S_InterferenceArmElevator2 :=  FaultSim(FaultLow:= VerificationBusyBlockedLow , FaultHigh := VerificationBusyBlockedHigh , Input := VerificationBusy);
S_IsElevatorUp2 :=  FaultSim(FaultLow:=CylinderUpToMeasureLoadBlockedLow  , FaultHigh := CylinderUpToMeasureLoadBlockedHigh , Input := CylinderUpToMeasureLoad);
S_IsElevatorDown2 :=  FaultSim(FaultLow:= CylinderDownToMeasureLoadBlockedLow , FaultHigh := CylinderDownToMeasureLoadBlockedHigh , Input := CylinderDownToMeasureLoad);
S_CylinderRetracted2 :=  FaultSim(FaultLow:= CylinderOfExtractionInRetroactivePositionBlockedLow , FaultHigh := CylinderOfExtractionInRetroactivePositionBlockedHigh , Input := CylinderOfExtractionInRetroactivePosition);
S_CylinderExtended2 :=  FaultSim(FaultLow:= ToExtendCylinderOfExtractionVsGuideBlocked , FaultHigh := ToExtendCylinderOfExtractionVsGuideBlockedHigh , Input := CylinderOfExtractionInExtensivePosition);
S_ElementInElevator2 :=  FaultSim(FaultLow:= ReadyLoadForVerificationBlockedLow , FaultHigh := ReadyLoadForVerificationBlockedHigh , Input := ReadyLoadForVerification);
S_Color2 :=  FaultSim(FaultLow:= ColourMeasurementBlockedLow , FaultHigh := ColourMeasurementBlockedHigh , Input := ColourMeasurement); (* 1 for silver-red element / 0 for black *)
S_IsHigh2 :=  FaultSim(FaultLow:= MeasurementNotOkBlockedLow , FaultHigh := MeasurementNotOkBlockedHigh , Input := MeasurementNotOk);(*1 for high element / 0 for short element*)

(*Sensors of the 3° station*)

S_RotaryAlligned3 :=  FaultSim(FaultLow:= AlignementRotaryTableWithPositioningsBlockedLow , FaultHigh := AlignementRotaryTableWithPositioningsBlockedHigh , Input := AlignementRotaryTableWithPositionings);
S_AvaiableElement3 :=  FaultSim(FaultLow:= AvailableLoadForWorkingStationBlockedLow , FaultHigh := AvailableLoadForWorkingStationBlockedHigh , Input := AvailableLoadForWorkingStation);
S_ControlElement3 :=  FaultSim(FaultLow:= AvailableLoadInControlPositioningBlockedLow , FaultHigh := AvailableLoadInControlPositioningBlockedHigh , Input := AvailableLoadInControlPositioning);
S_DrillElement3 :=  FaultSim(FaultLow:= AvailableLoadInDrillingPositioningBlockedLow , FaultHigh := AvailableLoadInDrillingPositioningBlockedHigh , Input := AvailableLoadInDrillingPositioning);
S_IsOnTheRightSide3 :=  FaultSim(FaultLow:= InControlLoadInWrongPositionToBeDrilledBlockedLow , FaultHigh := InControlLoadInWrongPositionToBeDrilledBlockedHigh , Input := InControlLoadInWrongPositionToBeDrilled);
S_DrillUp3 :=  FaultSim(FaultLow:= DrillingUnitUpBlockedLow , FaultHigh := DrillingUnitUpBlockedHigh , Input := DrillingUnitUp);
S_DrillDown3 :=  FaultSim(FaultLow:= DrillingUnitDownBlockedLow , FaultHigh := DrillingUnitDownBlockedHigh , Input := DrillingUnitDown);

(*Sensors of the 4° station*)

S_SpringCylinderExtended4 :=  FaultSim(FaultLow:= ToExtractSpringInAssemblyStationInExtensivePositionBlockedLow , FaultHigh := ToExtractSpringInAssemblyStationInExtensivePositionBlockedHigh , Input := ToExtractSpringInAssemblyStationInExtensivePosition);
S_SpringCylinderRetracted4 :=  FaultSim(FaultLow:= ToExtractSpringInAssemblyStationInRetroactivePositionBlockedLow , FaultHigh := ToExtractSpringInAssemblyStationInRetroactivePositionBlockedHigh , Input := ToExtractSpringInAssemblyStationInRetroactivePosition);
S_BlackPistonGiven4 :=  FaultSim(FaultLow:= PistonSelectorIsOnTheRightBlockedLow , FaultHigh := PistonSelectorIsOnTheRightBlockedHigh , Input := PistonSelectorIsOnTheRight);
S_SilverPistonGiven4 :=  FaultSim(FaultLow:= PistonSelectorIsOnTheLeftBlockedLow , FaultHigh := PistonSelectorIsOnTheLeftBlockedHigh , Input := PistonSelectorIsOnTheLeft);
S_NoCover4 :=  FaultSim(FaultLow:= EmptyCoverHouseInAssemblyStationBlockedLow , FaultHigh := EmptyCoverHouseInAssemblyStationBlockedHigh , Input := EmptyCoverHouseInAssemblyStation);
S_CoverCylinderRetracted4 :=  FaultSim(FaultLow:= ToExtractCoverInAssemblyStationInRetroactivePositionBlockedLow , FaultHigh := ToExtractCoverInAssemblyStationInRetroactivePositionBlockedHigh , Input := ToExtractCoverInAssemblyStationInRetroactivePosition);
S_CoverCylinderExtracted4 :=  FaultSim(FaultLow:= ToExtractCoverInAssemblyStationInExtensivePositionBlockedLow , FaultHigh := ToExtractCoverInAssemblyStationInExtensivePositionBlockedHigh , Input := ToExtractCoverInAssemblyStationInExtensivePosition);
S_ElementAvailable4 :=  FaultSim(FaultLow:= AvailableLoadForRobotBlockedLow , FaultHigh := AvailableLoadForRobotBlockedHigh , Input := AvailableLoadForRobot);

(*Robot sensors simulation*)

RobotInInitialPosition := Bit0Input AND Bit1Input;
RobotInAssemblyUnit := Bit3Input;
RobotInPistonWarehouse := Bit0Input AND NOT Bit1Input;
RobotInSpringWarehouse := NOT Bit0Input AND Bit1Input;
RobotInCoverWarehouse := Bit2Input;

S_RobotInInitial4 :=  FaultSim(FaultLow:= RobotInInitialPositionBlockedLow , FaultHigh := RobotInInitialPositionBlockedHigh , Input := RobotInInitialPosition);
S_RobotAssembly4 :=  FaultSim(FaultLow:= RobotInAssemblyUnitBlockedLow , FaultHigh := RobotInAssemblyUnitBlockedHigh , Input := RobotInAssemblyUnit);
S_RobotPiston4 :=  FaultSim(FaultLow:= RobotInPistonWarehouseBlockedLow , FaultHigh := RobotInPistonWarehouseBlockedHigh , Input := RobotInPistonWarehouse);
S_RobotSpring4 :=  FaultSim(FaultLow:= RobotInSpringWarehouseBlockedLow , FaultHigh := RobotInSpringWarehouseBlockedHigh , Input := RobotInSpringWarehouse);
S_RobotCover4 :=  FaultSim(FaultLow:= RobotInCoverWarehouseBlockedLow , FaultHigh := RobotInCoverWarehouseBlockedHigh , Input := RobotInCoverWarehouse);


(*Buttons*)

B_Start := Start;
B_Reset := Reset;
B_Freeze := NOT FreezeStopPuls;
B_Stop := NOT Stop;
B_Emergency := NOT EmergencyStop;
B_FullWarehouse := FullWarehouse;
B_OnlyBlackElement := ToWorkBlackLoad; (*1 to work only on black elements / 0 to work only on red/silver elements*)
B_AllColors := ToWorkBlackOrRedLoad; (*1 all colors / 0 only one color check B_OnlyBlackElement*)
B_FaultyElementRemoved := UpsideDownLoadRemovedInExpelling;
B_FillAll := FillAllWarehouses;
END_PROGRAM

(* POU Bridge/FaultSim, ST *)
FUNCTION FaultSim : BOOL

VAR_INPUT

	FaultLow: BOOL;
	FaultHigh: BOOL;
	Input: BOOL;

END_VAR

VAR
END_VAR
IF FaultLow THEN
	FaultSim := FALSE;
ELSIF FaultHigh THEN
	FaultSim := TRUE;
ELSE
	FaultSim := Input;
END_IF
END_FUNCTION

(* POU Main, ST *)
PROGRAM Main

VAR

	Stazione1: S1;
	Stazione2: S2;
	Stazione3: S3;
	Stazione4: S4;
	Lights: Lights;
	InitializationDone: BOOL := FALSE;
	ElementS2: CharacterisazionElement;
	ElementS3: CharacterisazionElement;
	ElementS4: CharacterisazionElement;
	OperationType: INT := INIT;
	Station1OperationType: INT := INIT;
	Station2OperationType: INT := INIT;
	Station3OperationType: INT := INIT;
	Station4OperationType: INT := INIT;
	NotSafeToRestart: BOOL;
	OnPhaseStopDone: BOOL;
	StopDone: BOOL;
	FirstPowerOn : BOOL := TRUE;
	RunCycles: INT := 0; (* Debug Variable used to take time-measurements *)

END_VAR
IF (OperationType = INIT) THEN
	SignHandlerOperationType := INIT;
ELSE
	SignHandlerOperationType := RUN;
END_IF

SignalHandler();

IF EmergencyInStop THEN

	OperationType := EMERGENCYSTOPMACHINE;
	Station1OperationType := IMMEDIATESTOPMACHINE; (*In emergency operation type Stations act as in the immediate stop case*)
	Station2OperationType := IMMEDIATESTOPMACHINE;
	Station3OperationType := IMMEDIATESTOPMACHINE;
	Station4OperationType := IMMEDIATESTOPMACHINE;
	Stazione1.StartButton := FALSE;

END_IF

CASE OperationType OF

	INIT:

		BridgeInitOperation := TRUE; (* Used only for Real Plant *)
		IF NOT MachineNOTOkForReset THEN		(* After a Reset it is FALSE, but not for first POWER-ON *)

			FirstPowerOn := FALSE;
			LightMachineToBeEmpty := FALSE;
			ButtonMachineToBeEmptyInvisible := TRUE;
			Station1OperationType := INIT;
			Station2OperationType := INIT;
			Station3OperationType := INIT;
			Station4OperationType := INIT;

		END_IF

		IF  Stazione1.InitializationDone1 AND  Stazione2.InitializationDone2 AND Stazione3.InitializationDone3  AND Stazione4.InitializationDone4  THEN (*Wait all station initialized*)
			InitializationDone:=TRUE;
			OperationType := READYTORUN;
		END_IF

	READYTORUN: (* Idle State*)

		BridgeInitOperation := FALSE; (* Used only for Real Plant *)
		Station1OperationType := READYTORUN;
		Station2OperationType := READYTORUN;
		Station3OperationType := READYTORUN;
		Station4OperationType := READYTORUN;

		IF B_Start THEN

			MachineNOTOkForReset := TRUE;
			LightMachineToBeEmpty := TRUE;
			OperationType:= RUN;
			Stazione1.StartButton := TRUE;

		END_IF

	RUN:

		RunCycles := RunCycles +1; (* For Diagnostic *)

		Station1OperationType := RUN;
		Station2OperationType := RUN;
		Station3OperationType := RUN;
		Station4OperationType := RUN;

		Stazione1.Go:= Stazione2.GoS1; (*To NOT have interference between stations *) (* Station(i+1) communicate when Station(i) can go i= 1,2,3 *)
		Stazione2.Go:= Stazione3.GoS2;
		Stazione3.Go:= Stazione4.GoS3;

		ElementS2.Color:=Stazione2.ActualColor;
		ElementS3.Over:=Stazione3.PieceOverturned;
		Stazione4.ElementColor:= ElementS4.Color;
		Stazione4.ElementOver:= ElementS4.Over;

		IF Stazione2.PassElementDefinition THEN (*Station(i) communicate the characterization of the piece done to Station(i+1) i= 2,3*)
			ElementS3.Color := ElementS2.Color;
		END_IF

		IF Stazione3.PassElementDefinition THEN
			ElementS4.Color := ElementS3.Color;
			ElementS4.Over := ElementS3.Over;
		END_IF

		IF ImmediateInStop THEN

			OperationType := IMMEDIATESTOPMACHINE;
			Station1OperationType := IMMEDIATESTOPMACHINE;
			Station2OperationType := IMMEDIATESTOPMACHINE;
			Station3OperationType := IMMEDIATESTOPMACHINE;
			Station4OperationType := IMMEDIATESTOPMACHINE;
			Stazione1.StartButton := FALSE;

		END_IF

		IF OnPhaseInStop THEN

			OperationType := ONPHASESTOPMACHINE;
			Station1OperationType := ONPHASESTOPMACHINE;
			Station2OperationType := ONPHASESTOPMACHINE;
			Station3OperationType := ONPHASESTOPMACHINE;
			Station4OperationType := ONPHASESTOPMACHINE;
			Stazione1.StartButton := FALSE;

		END_IF

	IMMEDIATESTOPMACHINE:

		IF NOT ImmediateInStop AND StopDone THEN  (* Wait until all the stations stop*)
			IF NotSafeToRestart  THEN
				OperationType := READYTORESET;
			ELSE
				OperationType := READYTORUN;
			END_IF
		END_IF


	ONPHASESTOPMACHINE:

		IF OnPhaseStopDone THEN (* Wait until all the stations stop*)
			OperationType := READYTORUN;
		END_IF

	EMERGENCYSTOPMACHINE:

		IF StopDone THEN (* Wait until all the stations stop*)
			OperationType := READYTORESET;
		END_IF

	READYTORESET:

		ButtonMachineToBeEmptyInvisible := FALSE;
		LightMachineToBeEmpty := TRUE;
		Station1OperationType := READYTORESET;
		Station2OperationType := READYTORESET;
		Station3OperationType := READYTORESET;
		Station4OperationType := READYTORESET;

		IF B_Reset AND NOT(ImmediateInStop OR EmergencyInStop OR NOT NoSignalsToReset OR MachineNOTOkForReset)  THEN
			InitializationDone := FALSE;
			OperationType := INIT;
		END_IF

END_CASE

AllStationsIdle := (	Stazione1.Idle AND Stazione2.Idle AND Stazione3.Idle AND Stazione4.Idle AND  (OperationType=RUN));	(* Signal Used to Stop Machine for inactivity*)
NotSafeToRestart := Stazione1.NotSafeToRestart OR Stazione2.NotSafeToRestart OR Stazione3.NotSafeToRestart OR Stazione4.NotSafeToRestart;
OnPhaseStopDone := Stazione1.OnPhaseStopDone1 AND Stazione2.OnPhaseStopDone2 AND Stazione3.OnPhaseStopDone3 AND Stazione4.OnPhaseStopDone4;
StopDone := Stazione1.StopDone1 AND Stazione2.StopDone2 AND Stazione3.StopDone3 AND Stazione4.StopDone4;

(*Update calls*)

ClocksGeneration.OperationType:= OperationType;
ClocksGeneration();

Lights.OperationType:= OperationType;
Lights.Element2.Color := ElementS2.Color;
Lights.Element3.Color := ElementS3.Color;
Lights.Element3.Over := Stazione3.PieceOverturned;
Lights.WriteLight2 := NOT Stazione2.GoS1;
Lights.WriteLight3 := Stazione3.WriteLight;
Lights.WriteLight4 := NOT Stazione4.Idle;
Lights.Element4 := Stazione4.Element;
Lights.InitializationDone:=InitializationDone;
Lights.RobotMoving := Stazione4.RobotIsMoving;
Lights.RobotOn := Stazione4.RobotIsOn;
Lights.PieceToDiscard2 := Stazione2.PieceToDiscard2;
Lights.Rejected:=Stazione4.Rejected;
Lights.Completed:=Stazione4.Completed;

 IF ClocksGeneration.Clock2ms AND NOT FirstPowerOn THEN
Lights();
Stazione1(OperationType := Station1OperationType);
Stazione2(OperationType := Station2OperationType);
Stazione3(OperationType := Station3OperationType);
Stazione4(OperationType := Station4OperationType);
 END_IF
END_PROGRAM

(* POU Work_Station/S1, ST *)
(* @OBJECTFLAGS := '0, 8' *)

FUNCTION_BLOCK S1

VAR_INPUT

	StartButton : BOOL;
	Go : BOOL;

END_VAR

VAR_OUTPUT

	InitializationDone1: BOOL;
	OnPhaseStopDone1: BOOL := FALSE;
	StopDone1: BOOL := FALSE;
	NotSafeToRestart: BOOL;
	Idle: BOOL;

END_VAR

VAR

	Cylinder: GenericDevice;
	Rotary : GenericDevice;
	Vacuum :GenericDevice;
	Expulsion :GenericDevice;
	EnableRotary: BOOL := FALSE;
	DisableRotary: BOOL:= FALSE;
	StateMachine: INT;
	EnableCylinder: BOOL := FALSE;
	DisableCylinder: BOOL := FALSE;
	EnableVacuum: BOOL := FALSE;
	DisableVacuum: BOOL := FALSE;
	EnableExpulsion: BOOL := FALSE;
	DisableExpulsion: BOOL := FALSE;
	NextElementReady: BOOL;
	CylinderInitialized: BOOL := FALSE;
	RotaryInitialized: BOOL := FALSE;
	VacuumInitialized: BOOL := FALSE;
	ExpulsionInitialized: BOOL := FALSE;
	ActivateVacuum: BOOL := FALSE;
	ActivateExpulsion: BOOL := FALSE;

END_VAR

VAR_IN_OUT

	OperationType: INT;

END_VAR
CASE OperationType OF

	INIT:

		IF CylinderInitialized AND RotaryInitialized AND VacuumInitialized AND ExpulsionInitialized THEN (* Wait until all devices are initialized*)
			InitializationDone1 := TRUE;
		END_IF

	READYTORUN:

		NotSafeToRestart := FALSE;
		OnPhaseStopDone1 := FALSE;
		StopDone1 := FALSE;

	RUN:

		IF ActivateVacuum THEN (*To safely restart after an immediate stop*)
			EnableVacuum := TRUE;
			ActivateVacuum := FALSE;
		END_IF

		IF ActivateExpulsion THEN (*To safely restart after an immediate stop*)
			EnableExpulsion := TRUE;
			ActivateExpulsion := FALSE;
		END_IF

		CASE StateMachine OF

			0: (*Wait Start button*)
				IF StartButton THEN
					StateMachine := 1;
				END_IF

			1:
				DisableCylinder := TRUE;
				StateMachine := 5;

			5: (*With no interference with the elevator the rotary can turn*)

				Idle:=TRUE;

				IF NOT DisableCylinder AND  NOT S_EmptyWarehouse1 AND Go THEN
					Idle:=FALSE;
					DisableRotary:=TRUE;
					StateMachine :=10;
				END_IF

			10: (*Moving the element with the cylinder*)

				IF NOT DisableRotary THEN
					EnableCylinder := TRUE;
					StateMachine := 15;
				END_IF

			15: (*Turn rotary*)

				IF NOT EnableCylinder  THEN
					EnableRotary := TRUE;
					StateMachine := 20;
				END_IF

			20: (*Activation vacuum*)

				IF NOT EnableRotary THEN
					EnableVacuum := TRUE;
					StateMachine := 25;
				END_IF

			25: (*Move Rotary to station 2 and cylinder retracts*)

				IF NOT EnableVacuum AND Go THEN
					DisableRotary := TRUE;
					DisableCylinder := TRUE;
					StateMachine := 30;
				END_IF

			30: (*Disable vacuum *)

				IF NOT DisableRotary AND  NOT DisableCylinder AND NOT ActivateVacuum THEN
					DisableVacuum := TRUE;
					IF NOT S_EmptyWarehouse1 THEN (*If there is a piece available the cylinder ejects it before enabling the rotary*)
						EnableCylinder:=TRUE;
						NextElementReady := TRUE;
					ELSE
						NextElementReady := FALSE;
					END_IF

					StateMachine := 35;
				END_IF

			35: (*Expell the element from the suction cup *)

				IF (NOT DisableVacuum AND NOT NextElementReady) OR (NOT DisableVacuum AND NOT EnableCylinder AND NextElementReady) THEN
					EnableExpulsion := TRUE;
					StateMachine := 40;
				END_IF

			40: (*Move  the rotary to warehouse*)

				IF NOT EnableExpulsion THEN
					DisableExpulsion:=TRUE;
					EnableRotary := TRUE;
					StateMachine := 50;
				END_IF

			50: (*Go back to the initial state*)

				IF NOT EnableRotary AND NOT DisableExpulsion THEN
					IF NextElementReady THEN
						StateMachine:=20;
					ELSE
						StateMachine := 5;
					END_IF
				END_IF

	END_CASE

	IMMEDIATESTOPMACHINE:

		CASE StateMachine OF
			0:
				StopDone1 := TRUE;

			1:
				StopDone1 := TRUE;

			5:
				IF NOT DisableCylinder THEN
					StopDone1 := TRUE;
				END_IF

			10:
				IF NOT DisableRotary THEN
					StopDone1 := TRUE;
				END_IF

			15:
				IF NOT EnableCylinder  THEN
					StopDone1 := TRUE;
				END_IF

			20:
				IF NOT EnableRotary THEN
					StopDone1 := TRUE;
				END_IF

			25:
				DisableVacuum := TRUE;
				ActivateVacuum := TRUE;
				StopDone1 := TRUE;

			30:
				IF NOT DisableRotary AND  NOT DisableCylinder THEN
					DisableVacuum := TRUE;
					StopDone1 := TRUE;
				END_IF

			35:
				IF (NOT DisableVacuum AND NOT NextElementReady) OR (NOT DisableVacuum AND NOT EnableCylinder AND NextElementReady) THEN
					StopDone1 := TRUE;
				END_IF

			40:
				DisableExpulsion := TRUE;
				ActivateExpulsion := TRUE;
				StopDone1 := TRUE;

			50:
				IF NOT EnableRotary AND NOT DisableExpulsion THEN
					StopDone1 := TRUE;
				END_IF

	END_CASE

	ONPHASESTOPMACHINE:

		CASE StateMachine OF

			0:
				OnPhaseStopDone1 := TRUE;

			1:
				OnPhaseStopDone1 := TRUE;

			5:
				IF NOT DisableCylinder THEN
					OnPhaseStopDone1 := TRUE;
				END_IF

			10:
				IF NOT DisableRotary THEN
					OnPhaseStopDone1 := TRUE;
				END_IF

			15:
				IF NOT EnableCylinder  THEN
					OnPhaseStopDone1 := TRUE;
				END_IF

			20:
				IF NOT EnableRotary THEN
					OnPhaseStopDone1 := TRUE;
				END_IF

			25:
				IF NOT EnableVacuum THEN
					OnPhaseStopDone1 := TRUE;
				END_IF

			30:
				IF NOT DisableRotary AND  NOT DisableCylinder THEN
					DisableVacuum := TRUE;
					OnPhaseStopDone1 := TRUE;
				END_IF

			35:
				IF (NOT DisableVacuum AND NOT NextElementReady) OR (NOT DisableVacuum AND NOT EnableCylinder AND NextElementReady) THEN
					OnPhaseStopDone1 := TRUE;
				END_IF

			40:
				IF NOT EnableExpulsion THEN
					OnPhaseStopDone1 := TRUE;
				END_IF

			50:
				IF NOT EnableRotary AND NOT DisableExpulsion THEN
					OnPhaseStopDone1 := TRUE;
				END_IF
	END_CASE


	READYTORESET:

		InitializationDone1 := FALSE;
		StateMachine := 0;
		ActivateVacuum := FALSE;
		ActivateExpulsion := FALSE;

END_CASE

(*Cylinder Generic Device*)

Cylinder(DeviceEnableRequest:=EnableCylinder ,DeviceDisableRequest := DisableCylinder);
A_Cylinder1 := Cylinder.EnableDevice;
Cylinder.DeviceEnabled  := S_CylinderExtended1;
Cylinder.DeviceDisabled := S_CylinderRetracted1;
Cylinder.DeviceType := DEVICE_WITH_SINGLE_ACTUATION OR DEVICE_WITH_DOUBLE_FEEDBACK;
Cylinder.DeviceClock := ClocksGeneration.Clock2ms;
Cylinder.DeviceDiagnosticsEnabled := TRUE;
Cylinder.DeviceDisableTime := 20;
Cylinder.DeviceEnablePreset := TRUE;
Cylinder.DeviceEnableTime := 20;
Cylinder.DeviceOperation := OperationType;
CylinderInitialized := NOT Cylinder.DeviceNotInitialized;
F_Cylinder1 := Cylinder.DeviceFault;
F_S_Cylinder1 := Cylinder.DeviceSensorFault;
F_A_Cylinder1 := Cylinder.DeviceActuatorFault;
FH_A_Cylinder1 := Cylinder.DeviceActuatorFaultHigh;
FL_A_Cylinder1 := Cylinder.DeviceActuatorFaultLow;
FH_DS_Cylinder1 := Cylinder.DeviceDisabledSensorFaultHigh;
FL_DS_Cylinder1 := Cylinder.DeviceDisabledSensorFaultLow;
FH_ES_Cylinder1 := Cylinder.DeviceEnabledSensorFaultHigh;
FL_ES_Cylinder1 := Cylinder.DeviceEnabledSensorFaultLow;

(*Rotary Generic Device*)

Rotary(DeviceEnableRequest:=EnableRotary ,DeviceDisableRequest := DisableRotary);
A_ArmToElevator1 := Rotary.DisableDevice;
A_ArmToWarehouse1 := Rotary.EnableDevice;
Rotary.DeviceEnabled := S_ArmInWarehouse1;
Rotary.DeviceDisabled := S_ArmInElevator1;
Rotary.DeviceType := DEVICE_WITH_DOUBLE_FEEDBACK  OR DEVICE_WITH_DOUBLE_ACTUATION;
Rotary.DeviceClock := ClocksGeneration.Clock2ms;
Rotary.DeviceDiagnosticsEnabled := TRUE;
Rotary.DeviceDisableTime := 20;
Rotary.DeviceEnablePreset := TRUE;
Rotary.DeviceEnableTime := 20;
Rotary.DeviceOperation := OperationType;
RotaryInitialized := NOT Rotary.DeviceNotInitialized;
F_Rotary1 := Rotary.DeviceFault;
F_S_Rotary1 := Rotary.DeviceSensorFault;
F_A_Rotary1 := Rotary.DeviceActuatorFault;
FL_EA_Rotary1 := Rotary.DeviceEnableActuatorFaultLow;
FH_EA_Rotary1 := Rotary.DeviceEnableActuatorFaultHigh;
FL_DA_Rotary1 := Rotary.DeviceDisableActuatorFaultLow;
FH_DA_Rotary1 := Rotary.DeviceDisableActuatorFaultHigh;
FH_ES_Rotary1 := Rotary.DeviceEnabledSensorFaultHigh;
FL_ES_Rotary1 := Rotary.DeviceEnabledSensorFaultLow;
FH_DS_Rotary1 := Rotary.DeviceDisabledSensorFaultHigh;
FL_DS_Rotary1 := Rotary.DeviceDisabledSensorFaultLow;

(*Vacuum Generic Device*)

Vacuum(DeviceEnableRequest:=EnableVacuum ,DeviceDisableRequest := DisableVacuum);
Vacuum.DeviceEnabled:= S_VacuumOk1;
A_Vacuum1 := Vacuum.EnableDevice;
Vacuum.DeviceType := DEVICE_WITH_SINGLE_ACTUATION OR DEVICE_WITH_ENABLE_FEEDBACK;
Vacuum.DeviceClock := ClocksGeneration.Clock2ms;
Vacuum.DeviceDiagnosticsEnabled := TRUE;
Vacuum.DeviceDisableTime := 10;
Vacuum.DeviceEnablePreset := FALSE;
Vacuum.DeviceEnableTime := 10;
Vacuum.DeviceOperation := OperationType;
VacuumInitialized := NOT Vacuum.DeviceNotInitialized;
F_Vacuum1 := Vacuum.DeviceFault;
F_S_Vacuum1 := Vacuum.DeviceSensorFault;
F_A_Vacuum1 := Vacuum.DeviceActuatorFault OR Vacuum.DeviceEnabledSensorFault	(* CHECK *);
FH_A_Vacuum1 := Vacuum.DeviceActuatorFaultHigh;
FL_A_Vacuum1 := Vacuum.DeviceEnabledSensorFault;
FH_S_Vacuum1 := Vacuum.DeviceSensorFaultHigh;
FL_S_Vacuum1 := Vacuum.DeviceSensorFaultLow;

(*Expulsion Generic Device*)

Expulsion(DeviceEnableRequest:=EnableExpulsion ,DeviceDisableRequest := DisableExpulsion);
A_AirVacuum1 := Expulsion.EnableDevice;
Expulsion.DeviceType := DEVICE_WITH_SINGLE_ACTUATION OR DEVICE_WITHOUT_FEEDBACK;
Expulsion.DeviceClock := ClocksGeneration.Clock2ms;
Expulsion.DeviceDiagnosticsEnabled := TRUE;
Expulsion.DeviceDisableTime := 10;
Expulsion.DeviceEnablePreset := FALSE;
Expulsion.DeviceEnableTime := 10;
Expulsion.DeviceOperation := OperationType;
ExpulsionInitialized := NOT Expulsion.DeviceNotInitialized;
F_Expulsion1 := Expulsion.DeviceFault;

(* THINK DIAGNOSIS *)

FH_A_Expulsion1 := Expulsion.DeviceActuatorFaultHigh;
FL_A_Expulsion1 := Expulsion.DeviceActuatorFaultLow;
END_FUNCTION_BLOCK

(* POU MyLibraries/GenericDevice, ST *)
FUNCTION_BLOCK GenericDevice

	VAR_INPUT

		DeviceEnableTime : UINT;
		DeviceDisableTime : UINT;
		DeviceEnabled : BOOL;
		DeviceDisabled : BOOL;
		DeviceClock : BOOL;
		DeviceType : BYTE;
		DeviceEnablePreset : BOOL;
		DeviceOperation : INT;
		DeviceDiagnosticsEnabled: BOOL;

END_VAR

	VAR_OUTPUT

		EnableDevice : BOOL;
		DisableDevice : BOOL;

		DeviceDisabledSensorFaultLow : BOOL;
		DeviceDisabledSensorFaultHigh : BOOL;
		DeviceEnabledSensorFaultLow: BOOL;
		DeviceEnabledSensorFaultHigh : BOOL;
		DeviceEnableActuatorFaultLow: BOOL;
		DeviceEnableActuatorFaultHigh : BOOL;
		DeviceDisableActuatorFaultLow : BOOL;
		DeviceDisableActuatorFaultHigh : BOOL;

		DeviceActuatorFaultHigh : BOOL;
		DeviceActuatorFaultLow : BOOL;
		DeviceSensorFaultHigh : BOOL;
		DeviceSensorFaultLow : BOOL;

		DeviceSensorFault : BOOL;
		DeviceActuatorFault : BOOL;
		DeviceFault : BOOL;
		DeviceDisabledSensorFault : BOOL;
		DeviceEnabledSensorFault : BOOL;
		(* End of Diagnostic Internal Variables *)

		DeviceNotInitialized : BOOL;

	END_VAR

	VAR_IN_OUT

		DeviceEnableRequest : BOOL;
		DeviceDisableRequest : BOOL;

	END_VAR

	VAR

		DeviceState : DeviceStateType := 0;
		DeviceTimer : UINT := 0;
		Timeout : BOOL;

	END_VAR

	VAR_EXTERNAL

	(*Feedback*)

	DEVICE_WITHOUT_FEEDBACK : BYTE := 2#01000000;
	DEVICE_WITH_ENABLE_FEEDBACK : BYTE := 2#00010000;
	DEVICE_WITH_DISABLE_FEEDBACK : BYTE := 2#00100000;
	DEVICE_WITH_DOUBLE_FEEDBACK : BYTE := 2#00110000;
	DEVICE_FEEDBACK_MASK : BYTE := 2#11110000;

	(*Actuation*)

	DEVICE_WITH_SINGLE_ACTUATION : BYTE := 2#00000001;
	DEVICE_WITH_DOUBLE_ACTUATION : BYTE := 2#00000011;
	DEVICE_WITH_DA_NO_RETAIN : BYTE := 2#00000010;
	DEVICE_ACTUATION_MASK : BYTE := 2#00001111;

	END_VAR
(*** DEVICE CLOCK HANDLER ***)

IF DeviceClock AND (DeviceTimer > 0) THEN

	DeviceTimer := DeviceTimer - 1;

END_IF;

Timeout := (DeviceTimer = 0);


(*** DEVICE INITIALIZATION HANDLER ***)

IF (DeviceOperation = INIT) THEN

	DeviceEnableRequest := FALSE;
	DeviceDisableRequest := FALSE;

	IF DeviceEnablePreset THEN
		EnableDevice := TRUE;
		DeviceTimer := DeviceEnableTime;

		IF (NOT (DeviceDisabled AND DeviceEnabled)) THEN
			DeviceState := DeviceEnablePhaseState;
		ELSE
			DeviceState := DeviceEnabledState;
		END_IF;
		DeviceNotInitialized := NOT DeviceEnabled OR DeviceDisabled;
	ELSE
		EnableDevice := FALSE;
		DeviceTimer := DeviceDisableTime;
		IF (NOT (DeviceDisabled AND DeviceEnabled)) THEN
			DeviceState := DeviceDisablePhaseState;
		ELSE
			DeviceState := DeviceDisabledState;
		END_IF;
		DeviceNotInitialized := DeviceEnabled OR NOT DeviceDisabled;
	END_IF;

	CASE (DeviceType AND DEVICE_FEEDBACK_MASK) OF

		DEVICE_WITH_ENABLE_FEEDBACK:
			DeviceDisabled := NOT DeviceEnabled;

		DEVICE_WITH_DISABLE_FEEDBACK :
			DeviceEnabled := NOT DeviceDisabled;

		DEVICE_WITHOUT_FEEDBACK:
			DeviceEnabled := DeviceEnablePreset;
			DeviceDisabled := NOT DeviceEnabled;

	END_CASE;

	CASE (DeviceType AND DEVICE_ACTUATION_MASK) OF

		DEVICE_WITH_DOUBLE_ACTUATION:
			DisableDevice := NOT EnableDevice;

		DEVICE_WITH_DA_NO_RETAIN: (* Not sure *)
			EnableDevice := EnableDevice AND (DeviceState = DeviceEnablePhaseState);
			DisableDevice := NOT EnableDevice AND (DeviceState = DeviceDisablePhaseState);

	END_CASE;
ELSE

	(*** DEVICE SENSORS HANDLER ***)

	(*Device with single actuation and single disable feedback*)

	IF (DeviceType AND DEVICE_FEEDBACK_MASK) = DEVICE_WITH_DISABLE_FEEDBACK THEN
		DeviceEnabled := NOT DeviceDisabled AND ((DeviceState = DeviceEnabledState) OR (DeviceState = DeviceEnablePhaseState) AND Timeout);
	END_IF;

	(*Device with single actuation and single enable feedback*)

	IF (DeviceType AND DEVICE_FEEDBACK_MASK) = DEVICE_WITH_ENABLE_FEEDBACK THEN
		DeviceDisabled := NOT DeviceEnabled AND ((DeviceState = DeviceDisabledState) OR (DeviceState = DeviceDisablePhaseState) AND Timeout);
	END_IF;

	(*Device with single actuation and NO feedback*)

	IF (DeviceType AND DEVICE_FEEDBACK_MASK) = DEVICE_WITHOUT_FEEDBACK THEN

		DeviceEnabled :=( (DeviceState = DeviceEnabledState) OR (DeviceState = DeviceEnablePhaseState)) AND Timeout;

		DeviceDisabled := (DeviceState = DeviceDisabledState) OR (DeviceState = DeviceDisablePhaseState) AND Timeout;

	END_IF;


	(*** DEVICE ACTUATORS HANDLER ***)

	(* Device with double actuation*)

	IF (DeviceType AND DEVICE_ACTUATION_MASK) = DEVICE_WITH_DOUBLE_ACTUATION THEN

		DisableDevice := NOT EnableDevice;

	END_IF;

	(* Device with double actuation and NO retain *)

	IF (DeviceType AND DEVICE_ACTUATION_MASK) = DEVICE_WITH_DA_NO_RETAIN THEN

		EnableDevice := EnableDevice AND (DeviceState = DeviceEnablePhaseState);

		DisableDevice := NOT EnableDevice AND (DeviceState = DeviceDisablePhaseState);

	END_IF;

END_IF;


(*** DEVICE CONTROL HANDLER ***)

CASE DeviceState OF

	DeviceDisabledState:

		DeviceDisableRequest := FALSE;

		IF DeviceEnableRequest THEN

			EnableDevice := TRUE;
			DeviceTimer := DeviceEnableTime;
			DeviceState := DeviceEnablePhaseState;

		END_IF;

	DeviceEnablePhaseState:

		IF DeviceDisableRequest THEN

			DeviceEnableRequest := FALSE;
			EnableDevice := FALSE;
			DeviceTimer := DeviceDisableTime;
			DeviceState := DeviceDisablePhaseState;

		END_IF;

		IF DeviceEnabled THEN

			DeviceEnableRequest := FALSE;
			DeviceTimer := 0;
			DeviceState := DeviceEnabledState;

		END_IF;

	DeviceEnabledState:

		DeviceEnableRequest := FALSE;

		IF DeviceDisableRequest THEN

			EnableDevice := FALSE;
			DeviceTimer := DeviceDisableTime;
			DeviceState := DeviceDisablePhaseState;

		END_IF;

	DeviceDisablePhaseState:

		IF DeviceEnableRequest THEN

			DeviceDisableRequest := FALSE;
			EnableDevice := TRUE;
			DeviceTimer := DeviceEnableTime;
			DeviceState := DeviceEnablePhaseState;

		END_IF;

		IF DeviceDisabled THEN

			DeviceDisableRequest := FALSE;
			DeviceTimer := 0;
			DeviceState := DeviceDisabledState;

		END_IF;

END_CASE;

(*** DEVICE DIAGNOSTICS HANDLER ***)

IF DeviceDiagnosticsEnabled THEN

	(* CHECKS HIGH/LOW FAULTS FOR DOUBLE FEEDBACK/ACTUATION TYPES **)

	DeviceDisabledSensorFaultLow := (NOT EnableDevice AND NOT DeviceDisabled AND NOT DeviceEnabled AND ((DeviceState=DeviceDisabledState) OR (DeviceState=DeviceDisablePhaseState))) AND Timeout;	(* FOR DOUBLE FEEDBACK TYPE *)
	DeviceDisabledSensorFaultHigh := (EnableDevice AND DeviceDisabled AND DeviceEnabled AND (DeviceState=DeviceEnabledState)) AND Timeout;					(* FOR DOUBLE FEEDBACK TYPE *)
	DeviceEnabledSensorFaultHigh := (NOT EnableDevice AND DeviceDisabled AND DeviceEnabled AND (DeviceState=DeviceDisabledState)) AND Timeout;				(* FOR DOUBLE FEEDBACK TYPE *)
	DeviceEnabledSensorFaultLow := (EnableDevice AND NOT DeviceDisabled AND NOT DeviceEnabled AND ((DeviceState=DeviceEnablePhaseState) OR (DeviceState=DeviceEnabledState)) ) AND Timeout;			(* FOR DOUBLE FEEDBACK TYPE *)

	DeviceEnableActuatorFaultLow := (EnableDevice AND DeviceDisabled AND NOT DeviceEnabled  AND (DeviceState = DeviceEnablePhaseState)) AND Timeout;		(* FOR DOUBLE ACTUATION TYPE *)
	DeviceEnableActuatorFaultHigh := (NOT EnableDevice AND NOT DeviceDisabled AND DeviceEnabled AND DeviceState = (DeviceDisabledState)) AND Timeout;		(* FOR DOUBLE ACTUATION TYPE *)
	DeviceDisableActuatorFaultLow := (NOT EnableDevice AND NOT DeviceDisabled AND DeviceEnabled AND DeviceState = (DeviceDisablePhaseState)) AND Timeout;	(* FOR DOUBLE ACTUATION TYPE *)
	DeviceDisableActuatorFaultHigh := (EnableDevice AND DeviceDisabled AND NOT DeviceEnabled  AND DeviceState = (DeviceEnabledState)) AND Timeout;				(* FOR DOUBLE ACTUATION TYPE *)

	(** CHECKS HIGH/LOW FAULTS FOR SINGLE ACTUATION/FEEDBACK TYPES **)

	IF (DeviceType AND DEVICE_FEEDBACK_MASK) = DEVICE_WITH_DISABLE_FEEDBACK THEN	(* FOR SINGLE DISABLE FEEDBACK TYPE *)
		DeviceSensorFaultLow := DeviceDisabledSensorFaultLow;
		DeviceSensorFaultHigh := DeviceDisabledSensorFaultHigh;
	END_IF

	IF (DeviceType AND DEVICE_FEEDBACK_MASK) = DEVICE_WITH_ENABLE_FEEDBACK THEN 	(* FOR SINGLE ENABLE FEEDBACK TYPE *)
		DeviceSensorFaultLow := DeviceEnabledSensorFaultLow;
		DeviceSensorFaultHigh := DeviceEnabledSensorFaultHigh;
	END_IF

	DeviceActuatorFaultHigh:= (NOT EnableDevice AND NOT DeviceDisabled AND DeviceEnabled AND ((DeviceState=DeviceDisablePhaseState) OR (DeviceState=DeviceDisabledState))) AND Timeout;	(* FOR SINGLE ACTUATION TYPE *)
	DeviceActuatorFaultLow:= (EnableDevice AND DeviceDisabled AND NOT DeviceEnabled AND ((DeviceState=DeviceEnablePhaseState) OR (DeviceState=DeviceEnabledState))) AND Timeout;		(* FOR SINGLE ACTUATION TYPE *)

	(* UPDATE GENERIC FAULT OUTPUT for SIGNAL MANAGMENT *)

	IF (DeviceType AND DEVICE_ACTUATION_MASK)= DEVICE_WITH_SINGLE_ACTUATION THEN
		DeviceActuatorFault := DeviceActuatorFaultHigh OR DeviceActuatorFaultLow;
	ELSE
		DeviceActuatorFault := (NOT	EnableDevice AND NOT DeviceDisabled AND DeviceEnabled OR EnableDevice AND DeviceDisabled AND NOT DeviceEnabled) AND Timeout;
	END_IF
	IF (DeviceType AND DEVICE_FEEDBACK_MASK) = DEVICE_WITH_DOUBLE_FEEDBACK THEN
		DeviceSensorFault := DeviceEnabledSensorFaultHigh OR DeviceEnabledSensorFaultLow OR DeviceDisabledSensorFaultHigh OR DeviceDisabledSensorFaultLow;
	ELSE
		DeviceSensorFault := DeviceSensorFaultHigh OR DeviceSensorFaultLow;
	END_IF

	(** GENERIC CHECK (by slides) IF DEVICE FAULT **)

	DeviceDisabledSensorFault := (NOT EnableDevice AND NOT DeviceDisabled AND NOT DeviceEnabled OR EnableDevice AND	DeviceDisabled AND	DeviceEnabled) 	AND Timeout;
	DeviceEnabledSensorFault :=	(NOT EnableDevice AND DeviceDisabled AND DeviceEnabled OR EnableDevice AND NOT DeviceDisabled AND NOT	DeviceEnabled) AND Timeout;

(*	DeviceSensorFault := (DeviceDisabledSensorFault OR DeviceEnabledSensorFault) ;	(* OK FOR DOUBLE  FEEDBACK *) *)

	DeviceActuatorFault := (NOT	EnableDevice AND NOT DeviceDisabled AND DeviceEnabled OR EnableDevice AND DeviceDisabled AND NOT DeviceEnabled) AND Timeout;		(* OK FOR DOUBLE  ACTUATION *)

	DeviceFault := DeviceDisabledSensorFault OR DeviceEnabledSensorFault OR DeviceActuatorFault;

END_IF;
END_FUNCTION_BLOCK

(* POU MyLibraries/ClocksGeneration, ST *)
PROGRAM ClocksGeneration

VAR_INPUT

	OperationType: INT;

END_VAR

VAR_OUTPUT

 Clock2ms : BOOL;
 Clock10ms : BOOL;
 Clock100ms : BOOL;
 Clock1s : BOOL;

END_VAR


VAR

 SystemClock : BOOL;
 SystemClockOld : BOOL;
 TimerClock10ms : INT;
 TimerClock100ms : INT;
 TimerClock1s : INT;
 InitDone : BOOL := FALSE;

END_VAR
IF (OperationType = INIT) THEN
	IF NOT InitDone THEN
		SystemClockOld := TRUE;
		TimerClock10ms := 5;	(* Because we have edge_pos every 2 cycles *)
		TimerClock100ms := 10;
		TimerClock1s := 10;
		InitDone := TRUE;
	END_IF
ELSE
	InitDone := FALSE;
END_IF

SystemClock := NOT SystemClock;

Clock2ms := SystemClock;


IF Clock2ms THEN
	TimerClock10ms := TimerClock10ms -1 ;
END_IF

Clock10ms := (TimerClock10ms = 0);
IF Clock10ms THEN
	TimerClock10ms := 10;
	TimerClock100ms := TimerClock100ms - 1;
END_IF

Clock100ms := (TimerClock100ms = 0);
IF Clock100ms THEN
	TimerClock100ms := 10;
	TimerClock1s := TimerClock1s - 1;
END_IF

Clock1s := (TimerClock1s = 0);
IF Clock1s THEN
	TimerClock1s := 10;
END_IF
END_PROGRAM

(* POU Work_Station/S2, ST *)
(* @OBJECTFLAGS := '0, 8' *)

FUNCTION_BLOCK S2

VAR_INPUT

	Go:BOOL;

END_VAR
VAR_OUTPUT

	InitializationDone2: BOOL := FALSE;
	GoS1: BOOL;
	ActualColor:BOOL;
	PassElementDefinition: BOOL:=FALSE;
	OnPhaseStopDone2: BOOL := FALSE;
	StopDone2: BOOL;
	NotSafeToRestart: BOOL;
	PiecetoDiscard2 :BOOL := FALSE;
	Idle:BOOL;

END_VAR

VAR

	StateMachine: INT;
	Elevator: GenericDevice;
	EnableElevator: BOOL := FALSE;
	DisableElevator: BOOL := FALSE;
	Cylinder: GenericDevice;
	EnableCylinder: BOOL := FALSE;
	DisableCylinder: BOOL := FALSE;
	Air: GenericDevice;
	EnableAir: BOOL := FALSE;
	DisableAir: BOOL := FALSE;
	ActualHeight: BOOL;
	ElevatornInitialized: BOOL := FALSE;
	CylinderInitialized: BOOL := FALSE;
	AirInitialized: BOOL := FALSE;
	ActivateAir: BOOL := FALSE;

END_VAR

VAR_IN_OUT

	OperationType: INT;

END_VAR
CASE OperationType OF

	INIT:

		GoS1 := TRUE;
		IF ElevatornInitialized AND CylinderInitialized AND AirInitialized  THEN
			InitializationDone2:=TRUE;
		END_IF

	READYTORUN:

		NotSafeToRestart := FALSE;
		StopDone2 := FALSE;
		OnPhaseStopDone2 := FALSE;

	RUN:

		IF ActivateAir  THEN (*To safely restart after an immediate stop*)
			EnableAir := TRUE;
			ActivateAir := FALSE;
		END_IF

		CASE StateMachine OF

			0: (*Wait element and check color*)

				GoS1:=TRUE;
				PassElementDefinition:=FALSE;
				Idle:=TRUE;
				IF NOT S_InterferenceArmElevator2 AND S_ElementInElevator2 THEN
					GoS1:=FALSE;
					ActualColor:=S_Color2; (*red if true, black otherwise*)
					Idle:=FALSE;
					StateMachine := 5;
				END_IF

			5:(*Color Verification*)

				IF B_AllColors OR (B_OnlyBlackElement AND NOT S_Color2) OR (NOT B_OnlyBlackElement AND S_Color2) THEN (*Set from the switchboard*)
					StateMachine := 10;
				ELSE
					EnableCylinder := TRUE;
					StateMachine := 35;
				END_IF

			10: (*Elevator go up*)

				EnableElevator:=TRUE;
				StateMachine := 15;
		
			15: (*Check height*)

				IF NOT EnableElevator THEN
					ActualHeight := S_IsHigh2; (*high if true, low otherwise*)
					StateMachine := 20;
				END_IF
		
			20: (*Check good element or not*)

				IF (ActualColor XOR ActualHeight) THEN (*testing result NOT OK*)
					PieceToDiscard2 := TRUE;
					StateMachine := 25;
				ELSE (*testing result OK*)
					StateMachine := 100;
				END_IF
		
			(*PROCEDURE TO EXPELL WRONG ELEMENTS*)

			25:(*Elevator go down*)

				DisableElevator := TRUE;
				StateMachine := 30;
		
			30: (*Expell rejected element*)

				IF NOT DisableElevator THEN
					EnableCylinder := TRUE;
					StateMachine := 35;
				END_IF
		
			35: (*Disable cylinder*)

				IF NOT EnableCylinder THEN
					DisableCylinder := TRUE;
					StateMachine := 40;
				END_IF
		
			40: (*wait return of the cylinder*)

				IF NOT DisableCylinder THEN
					PieceToDiscard2 := FALSE;
					StateMachine := 0;
				END_IF
		
		
			(*PROCEDURE TO EXPELL GOOD ELEMENTS*)

			100: (*Enable slide air*)

				IF go THEN
					EnableAir := TRUE;
					StateMachine := 105;
				END_IF
		
			105: (*Expell good element and say the characteristics of the element to the next station*)

				IF NOT EnableAir THEN
					PassElementDefinition:=TRUE;
					EnableCylinder := TRUE;
					StateMachine := 110;
				END_IF
		
			110: (*Disable cylinder*)

				IF NOT EnableCylinder AND NOT ActivateAir THEN
					DisableCylinder:=TRUE;
					StateMachine := 115;
				END_IF
		
			115: (*Disable air and elevator go down*)

				IF NOT DisableCylinder THEN
					DisableAir:=TRUE;
					DisableElevator:=TRUE;
					StateMachine:= 120;
				END_IF
		
			120: (*Go back to initial state*)

				IF NOT DisableElevator THEN
					StateMachine := 0;
				END_IF

		END_CASE

	IMMEDIATESTOPMACHINE:

		CASE StateMachine OF

			0:
				StopDone2 := TRUE;
		
			10:
				StopDone2 := TRUE;

			15:
				IF NOT EnableElevator THEN
					StopDone2 := TRUE;
				END_IF
		
			20:
				StopDone2 := TRUE;

			25:
				StopDone2 := TRUE;

			30:
				IF NOT DisableElevator THEN
					StopDone2 := TRUE;
				END_IF
		
			35:
				IF NOT EnableCylinder THEN
					StopDone2 := TRUE;
				END_IF

			40:
				IF NOT DisableCylinder THEN
					StopDone2 := TRUE;
				END_IF

			100:
				StopDone2 := TRUE;
		
			105:
				DisableAir := TRUE;
				ActivateAir := TRUE;
				StopDone2 := TRUE;

			110:
				DisableAir := TRUE;
				ActivateAir := TRUE;
				IF NOT EnableCylinder THEN
					StopDone2 := TRUE;
				END_IF
		
			115:
				DisableAir := TRUE;
				IF NOT DisableCylinder THEN
					StopDone2 := TRUE;
				END_IF

			120:
				IF NOT DisableElevator THEN
					StopDone2 := TRUE;
				END_IF

		END_CASE

	ONPHASESTOPMACHINE:

		CASE StateMachine OF

			0:
				OnPhaseStopDone2 := TRUE;
		
			10:
				OnPhaseStopDone2 := TRUE;

			15:
				IF NOT EnableElevator THEN
					OnPhaseStopDone2 := TRUE;
				END_IF
		
			20:
				OnPhaseStopDone2 := TRUE;

			25:
				OnPhaseStopDone2 := TRUE;

			30:
				IF NOT DisableElevator THEN
					OnPhaseStopDone2 := TRUE;
				END_IF
		
			35:
				IF NOT EnableCylinder THEN
					OnPhaseStopDone2 := TRUE;
				END_IF
		
			40:
				IF NOT DisableCylinder THEN
					OnPhaseStopDone2 := TRUE;
				END_IF

			100:
				OnPhaseStopDone2 := TRUE;
		
			105:
				IF NOT EnableAir THEN
					OnPhaseStopDone2 := TRUE;
				END_IF

			110:
				IF NOT EnableCylinder THEN
					OnPhaseStopDone2 := TRUE;
				END_IF
		
			115:
				IF NOT DisableCylinder THEN
					OnPhaseStopDone2 := TRUE;
				END_IF

			120:
				IF NOT DisableElevator THEN
					OnPhaseStopDone2 := TRUE;
				END_IF

		END_CASE

	READYTORESET:

		InitializationDone2 := FALSE;
		StateMachine := 0;
		ActivateAir := FALSE;

END_CASE

(*Elevator Generic Device*)

Elevator(DeviceEnableRequest:=EnableElevator ,DeviceDisableRequest := DisableElevator);
A_ElevatorDown2 := Elevator.DisableDevice;
A_ElevatorUp2 := Elevator.EnableDevice;
Elevator.DeviceEnabled := S_IsElevatorUp2;
Elevator.DeviceDisabled := S_IsElevatorDown2;
Elevator.DeviceType := DEVICE_WITH_DOUBLE_FEEDBACK  OR DEVICE_WITH_DOUBLE_ACTUATION;
Elevator.DeviceClock := ClocksGeneration.Clock2ms;
Elevator.DeviceDiagnosticsEnabled := TRUE;
Elevator.DeviceDisableTime := 70;
Elevator.DeviceEnablePreset := FALSE;
Elevator.DeviceEnableTime := 50;
Elevator.DeviceOperation := OperationType;
ElevatornInitialized := NOT Elevator.DeviceNotInitialized;
F_Elevator2 := Elevator.DeviceFault;
F_S_Elevator2 := Elevator.DeviceSensorFault;
F_A_Elevator2 := Elevator.DeviceActuatorFault;
FH_EA_Elevator2 := Elevator.DeviceEnableActuatorFaultHigh;
FL_EA_Elevator2 := Elevator.DeviceEnableActuatorFaultLow;
FH_DA_Elevator2 := Elevator.DeviceDisableActuatorFaultHigh;
FL_DA_Elevator2 := Elevator.DeviceDisableActuatorFaultLow;
FH_ES_Elevator2 := Elevator.DeviceEnabledSensorFaultHigh;
FL_ES_Elevator2 := Elevator.DeviceEnabledSensorFaultLow;
FH_DS_Elevator2 := Elevator.DeviceDisabledSensorFaultHigh;
FL_DS_Elevator2 := Elevator.DeviceDisabledSensorFaultLow;

(*Cylinder Generic Device*)

Cylinder(DeviceEnableRequest:=EnableCylinder ,DeviceDisableRequest := DisableCylinder);
A_Cylinder2 := Cylinder.EnableDevice;
Cylinder.DeviceDisabled := S_CylinderRetracted2;
Cylinder.DeviceType := DEVICE_WITH_SINGLE_ACTUATION OR DEVICE_WITH_DISABLE_FEEDBACK;
Cylinder.DeviceClock := ClocksGeneration.Clock2ms;
Cylinder.DeviceDiagnosticsEnabled := TRUE;
Cylinder.DeviceDisableTime := 20;
Cylinder.DeviceEnablePreset := FALSE;
Cylinder.DeviceEnableTime := 20;
Cylinder.DeviceOperation := OperationType;
CylinderInitialized := NOT Cylinder.DeviceNotInitialized;
F_Cylinder2 := Cylinder.DeviceFault;
F_S_Cylinder2 := Cylinder.DeviceSensorFault;
F_A_Cylinder2 := Cylinder.DeviceActuatorFault;
FH_A_Cylinder2 := Cylinder.DeviceActuatorFaultHigh;
FL_A_Cylinder2 := Cylinder.DeviceActuatorFaultLow ;
FH_S_Cylinder2 := Cylinder.DeviceSensorFaultHigh;
FL_S_Cylinder2 := Cylinder.DeviceSensorFaultLow;

(*Air Generic Device*)

Air(DeviceEnableRequest:=EnableAir ,DeviceDisableRequest := DisableAir);
A_AirSlider2 :=  Air.EnableDevice;
Air.DeviceType := DEVICE_WITH_SINGLE_ACTUATION OR DEVICE_WITHOUT_FEEDBACK;
Air.DeviceClock := ClocksGeneration.Clock2ms;
Air.DeviceDiagnosticsEnabled := TRUE;
Air.DeviceDisableTime := 10;
Air.DeviceEnablePreset := FALSE;
Air.DeviceEnableTime := 10;
Air.DeviceOperation := OperationType;
AirInitialized := NOT Air.DeviceNotInitialized;
F_Air2 := Air.DeviceFault;

(* THINK DIAGNOSIS *)

FH_A_Air2 := Air.DeviceActuatorFaultHigh;
FL_A_Air2 := Air.DeviceActuatorFaultLow;
END_FUNCTION_BLOCK

(* POU Work_Station/S3, ST *)
FUNCTION_BLOCK S3

VAR_INPUT

	Go:BOOL;

END_VAR

VAR_OUTPUT

	InitializationDone3: BOOL := FALSE;
	GoS2 :BOOL:=FALSE;
	PieceOverturned: BOOL := FALSE;
	PassElementDefinition: BOOL := FALSE;
	NotSafeToRestart: BOOL;
	OnPhaseStopDone3: BOOL := FALSE;
	StopDone3: BOOL;
	WriteLight: BOOL;
	Idle:BOOL;

END_VAR

VAR

	Rotary: GenericDevice;
	DisableRotary: BOOL:=FALSE;
	Cylinder: GenericDevice;
	Drilling: GenericDevice;
	EnableDrilling: BOOL := FALSE;
	DisableDrilling: BOOL := FALSE;
	DrillCylinder: GenericDevice;
	EnableDrillCylinder: BOOL := FALSE;
	DisableDrillCylinder: BOOL := FALSE;
	Block: GenericDevice;
	EnableBlock: BOOL := FALSE;
	DisableBlock: BOOL := FALSE;
	Expell: GenericDevice;
	EnableExpell: BOOL := FALSE;
	DisableExpell: BOOL := FALSE;
	StateMachine: INT;
	EnableCylinder: BOOL := FALSE;
	DisableCylinder: BOOL := FALSE;
	EnableRotary: BOOL := FALSE;

	CylinderInitialized: BOOL := FALSE;
	DrillCylinderInitialized: BOOL := FALSE;
	DrillingInitialized: BOOL := FALSE;
	BlockInitialized: BOOL := FALSE;
	ExpellInitialized: BOOL := FALSE;

	StateMachineInit: INT;

END_VAR

VAR_IN_OUT

	OperationType: INT;

END_VAR
CASE OperationType OF

	INIT:

		GoS2 := TRUE;

		CASE StateMachineInit OF

			0:

				EnableRotary := TRUE;
				StateMachineInit := 1;

			1:

				IF S_RotaryAlligned3 THEN  (*Manual initialization of the rotary*)
					DisableRotary := TRUE;
					StateMachineInit := 2;
				END_IF

			2:

				IF NOT DisableRotary AND CylinderInitialized AND DrillCylinderInitialized AND DrillingInitialized AND BlockInitialized AND ExpellInitialized THEN
					InitializationDone3 := TRUE;
				END_IF

		END_CASE

	READYTORUN:

		NotSafeToRestart := FALSE;
		OnPhaseStopDone3 := FALSE;
		StopDone3 := FALSE;

	RUN:

		CASE StateMachine OF

			0: (*Wait for an available element*)

				GoS2:=TRUE;
				PassElementDefinition:=FALSE;
				WriteLight:=FALSE;
				Idle:=TRUE;
				IF S_AvaiableElement3 THEN
					GoS2 := FALSE;
					EnableRotary:=TRUE;
					PieceOverturned:=FALSE;
					Idle:=FALSE;
					StateMachine:=8;
				END_IF
		
			8: (* Wait for the allignment of the rotary*)

				IF NOT EnableRotary AND S_RotaryAlligned3 THEN
					DisableRotary := TRUE;
					StateMachine := 10;
				END_IF

			10: (* Enable control cylinder*)

				IF  NOT DisableRotary AND S_ControlElement3 THEN
					EnableCylinder:=TRUE;
					StateMachine :=15;
				END_IF

			15: (* Control if the piece is overturned*)

				IF NOT EnableCylinder THEN
					IF NOT S_IsOnTheRightSide3 THEN
						PieceOverturned:=TRUE;
					END_IF
					WriteLight:=TRUE;
					DisableCylinder:=TRUE;
					StateMachine:=20;
				END_IF
		
			20: (*Enable rotary*)

				IF NOT DisableCylinder THEN
					EnableRotary:=TRUE;
					StateMachine:=22;
				END_IF
		
			22: (* Wait for the allignment of the rotary*)

				IF NOT EnableRotary AND S_RotaryAlligned3 THEN
					DisableRotary := TRUE;
					StateMachine := 25;
				END_IF
		
			25: (*Drilling Station up to state 45*)

				IF NOT DisableRotary THEN
					IF PieceOverturned THEN
						EnableRotary:=TRUE;
						StateMachine:=52;
					ELSE
						EnableBlock:=TRUE;
						StateMachine:=30;
					END_IF
				END_IF
		
			30:

				IF NOT EnableBlock THEN
					EnableDrilling:=TRUE;
					StateMachine:=35;
				END_IF

			35:

				IF NOT EnableDrilling THEN
					EnableDrillCylinder:=TRUE;
					StateMachine:=40;
				END_IF

			40:

				IF NOT EnableDrillCylinder THEN
					DisableDrillCylinder:=TRUE;
					StateMachine:=45;
				END_IF
		
			45:

				IF NOT DisableDrillCylinder  THEN
					DisableDrilling:=TRUE;
					DisableBlock:=TRUE;
					StateMachine:=50;
				END_IF
		
			50: (*Enable rotary*)

				IF NOT DisableDrilling AND NOT DisableBlock THEN
					EnableRotary:=TRUE;
					StateMachine:=52;
				END_IF
		
			52: (* Wait for the allignment of the rotary*)

				IF NOT EnableRotary AND S_RotaryAlligned3 THEN
					DisableRotary := TRUE;
					StateMachine := 55;
				END_IF
		
			55: (*Expell element*)

				IF NOT DisableRotary  AND Go THEN
					PassElementDefinition:=TRUE;
					EnableExpell:=TRUE;
					StateMachine:=60;
				END_IF
		
			60:(*Disable expell cylinder*)

				IF NOT EnableExpell THEN
					DisableExpell:=TRUE;
					StateMachine:=65;
				END_IF
		
			65: (*Return to initial state*)

				IF NOT DisableExpell THEN
					StateMachine:=0;
				END_IF

		END_CASE

	IMMEDIATESTOPMACHINE:

		CASE StateMachine OF

			0:
				StopDone3 := TRUE;

			8:
				DisableRotary := TRUE;
				StopDone3 := TRUE;
				IF NOT S_RotaryAlligned3 THEN
					NotSafeToRestart := TRUE;
				END_IF

			10:
				IF NOT DisableRotary THEN
					StopDone3 := TRUE;
				END_IF
		
			15:
				IF NOT EnableCylinder THEN
					StopDone3 := TRUE;
				END_IF
		
			20:
				IF NOT DisableCylinder THEN
					StopDone3 := TRUE;
				END_IF
		
			22:
				DisableRotary := TRUE;
				StopDone3 := TRUE;
				IF NOT S_RotaryAlligned3 THEN
					NotSafeToRestart := TRUE;
				END_IF

			25:
				IF NOT DisableRotary THEN
					StopDone3 := TRUE;
				END_IF
		
			30:
				IF NOT EnableBlock THEN
					StopDone3 := TRUE;
				END_IF
		
			35:
				DisableDrilling := TRUE;
				NotSafeToRestart := TRUE;
				StopDone3 := TRUE;

			40:
				DisableDrilling := TRUE;
				NotSafeToRestart := TRUE;
				IF NOT EnableDrillCylinder THEN
					StopDone3 := TRUE;
				END_IF
		
			45:
				DisableDrilling := TRUE;
				NotSafeToRestart := TRUE;
				IF NOT DisableDrillCylinder THEN
					StopDone3 := TRUE;
				END_IF

			50:
				IF NOT DisableDrilling AND NOT DisableBlock THEN
					StopDone3 := TRUE;
				END_IF
		
			52:
				DisableRotary := TRUE;
				StopDone3 := TRUE;
				IF NOT S_RotaryAlligned3 THEN
					NotSafeToRestart := TRUE;
				END_IF

			55:
				IF NOT DisableRotary THEN
					StopDone3 := TRUE;
				END_IF

			60:
				IF NOT EnableExpell THEN
					StopDone3 := TRUE;
				END_IF
		
			65:
				IF NOT DisableExpell THEN
					StopDone3 := TRUE;
				END_IF

		END_CASE

	ONPHASESTOPMACHINE:

		CASE StateMachine OF

			0:
				OnPhaseStopDone3 := TRUE;
		
			8:
				IF NOT EnableRotary AND S_RotaryAlligned3 THEN
					DisableRotary := TRUE;
					StateMachine := 10;
				END_IF

			10:
				IF  NOT DisableRotary AND S_ControlElement3 THEN
					OnPhaseStopDone3 := TRUE;
				END_IF
		
			15:
				IF NOT EnableCylinder THEN
					OnPhaseStopDone3 := TRUE;
				END_IF
		
			20:
				IF NOT DisableCylinder THEN
					OnPhaseStopDone3 := TRUE;
				END_IF
		
			22:
				IF NOT EnableRotary AND S_RotaryAlligned3 THEN
					DisableRotary := TRUE;
					StateMachine := 25;
				END_IF
		
			25:
				IF NOT DisableRotary THEN
					OnPhaseStopDone3 := TRUE;
				END_IF
		
			30:
				IF NOT EnableBlock THEN
					OnPhaseStopDone3 := TRUE;
				END_IF
		
			35:
				IF NOT EnableDrilling THEN
					OnPhaseStopDone3 := TRUE;
				END_IF
		
			40:
				IF NOT EnableDrillCylinder THEN
					OnPhaseStopDone3 := TRUE;
				END_IF
		
			45:
				IF NOT DisableDrillCylinder THEN
					OnPhaseStopDone3 := TRUE;
				END_IF

			50:
				IF NOT DisableDrilling AND NOT DisableBlock THEN
					OnPhaseStopDone3 := TRUE;
				END_IF
		
			52:
				IF NOT EnableRotary AND S_RotaryAlligned3 THEN
					DisableRotary := TRUE;
					StateMachine := 55;
				END_IF
		
			55:
				IF NOT DisableRotary  AND Go THEN
					OnPhaseStopDone3 := TRUE;
				END_IF

			60:
				IF NOT EnableExpell THEN
					OnPhaseStopDone3 := TRUE;
				END_IF
		
			65:
				IF NOT DisableExpell THEN
					OnPhaseStopDone3 := TRUE;
				END_IF

		END_CASE

	READYTORESET:

		InitializationDone3 := FALSE;
		StateMachine := 0;
		StateMachineInit := 0;

END_CASE

(*Rotary table Generic Device*)

Rotary(DeviceEnableRequest:=EnableRotary ,DeviceDisableRequest := DisableRotary);
A_RotaryTable3 := Rotary.EnableDevice;
Rotary.DeviceDisabled := S_RotaryAlligned3;
Rotary.DeviceType := DEVICE_WITH_SINGLE_ACTUATION OR DEVICE_WITH_DISABLE_FEEDBACK;
Rotary.DeviceClock := ClocksGeneration.Clock2ms;
Rotary.DeviceDiagnosticsEnabled := TRUE;
Rotary.DeviceDisableTime := 20;
Rotary.DeviceEnablePreset := FALSE;
Rotary.DeviceEnableTime := 1;
Rotary.DeviceOperation := RUN;
F_RotaryTable3 := Rotary.DeviceFault;
F_S_RotaryTable3 := Rotary.DeviceSensorFault;
F_A_RotaryTable3 := Rotary.DeviceActuatorFault;
FH_A_RotaryTable3 := Rotary.DeviceActuatorFaultHigh;
FL_A_RotaryTable3 := Rotary.DeviceActuatorFaultLow;
FH_S_RotaryTable3 := Rotary.DeviceSensorFaultHigh;
FL_S_RotaryTable3 := Rotary.DeviceSensorFaultLow;


(*Check Cylinder Generic Device*)

Cylinder(DeviceEnableRequest:=EnableCylinder ,DeviceDisableRequest := DisableCylinder);
A_GoControl3 := Cylinder.EnableDevice;
Cylinder.DeviceType := DEVICE_WITH_SINGLE_ACTUATION OR DEVICE_WITHOUT_FEEDBACK;
Cylinder.DeviceClock := ClocksGeneration.Clock2ms;
Cylinder.DeviceDiagnosticsEnabled := TRUE;
Cylinder.DeviceDisableTime := 20;
Cylinder.DeviceEnablePreset := FALSE;
Cylinder.DeviceEnableTime := 20;
Cylinder.DeviceOperation := OperationType;
CylinderInitialized := NOT Cylinder.DeviceNotInitialized;
F_Cylinder3 := Cylinder.DeviceFault;

(* THINK DIAGNOSIS *)

FH_A_Cylinder3 := Cylinder.DeviceActuatorFaultHigh;
FL_A_Cylinder3 := Cylinder.DeviceActuatorFaultLow;


(*Drill Cylinder Generic Device*)

DrillCylinder(DeviceEnableRequest:=EnableDrillCylinder ,DeviceDisableRequest := DisableDrillCylinder);
A_ReturnDrill3 := DrillCylinder.DisableDevice;
A_GoDrill3 := DrillCylinder.EnableDevice;
DrillCylinder.DeviceEnabled := S_DrillDown3 ;
DrillCylinder.DeviceDisabled := S_DrillUp3 ;
DrillCylinder.DeviceType := DEVICE_WITH_DOUBLE_FEEDBACK  OR DEVICE_WITH_DOUBLE_ACTUATION;
DrillCylinder.DeviceClock := ClocksGeneration.Clock2ms;
DrillCylinder.DeviceDiagnosticsEnabled := TRUE;
DrillCylinder.DeviceDisableTime := 10;
DrillCylinder.DeviceEnablePreset := FALSE;
DrillCylinder.DeviceEnableTime := 10;
DrillCylinder.DeviceOperation := OperationType;
DrillCylinderInitialized := NOT DrillCylinder.DeviceNotInitialized;
F_DrillCylinder3 := DrillCylinder.DeviceFault;
F_S_DrillCylinder3 := DrillCylinder.DeviceSensorFault;
F_A_DrillCylinder3 := DrillCylinder.DeviceActuatorFault;
FH_EA_DrillCylinder3 := DrillCylinder.DeviceDisableActuatorFaultLow;
FL_EA_DrillCylinder3 := DrillCylinder.DeviceDisableActuatorFaultHigh;
FH_DA_DrillCylinder3 := DrillCylinder.DeviceEnableActuatorFaultLow;
FL_DA_DrillCylinder3 := DrillCylinder.DeviceEnableActuatorFaultHigh;
FH_ES_DrillCylinder3 := DrillCylinder.DeviceEnabledSensorFaultHigh;
FL_ES_DrillCylinder3 := DrillCylinder.DeviceEnabledSensorFaultLow;
FH_DS_DrillCylinder3 := DrillCylinder.DeviceDisabledSensorFaultHigh;
FL_DS_DrillCylinder3 := DrillCylinder.DeviceDisabledSensorFaultLow;


(*Drilling action Generic Device*)

Drilling(DeviceEnableRequest:=EnableDrilling ,DeviceDisableRequest := DisableDrilling);
A_Drilling3 := Drilling.EnableDevice;
Drilling.DeviceType := DEVICE_WITH_SINGLE_ACTUATION OR DEVICE_WITHOUT_FEEDBACK;
Drilling.DeviceClock := ClocksGeneration.Clock2ms;
Drilling.DeviceDiagnosticsEnabled := TRUE;
Drilling.DeviceDisableTime := 20;
Drilling.DeviceEnablePreset := FALSE;
Drilling.DeviceEnableTime := 20;
Drilling.DeviceOperation := OperationType;
DrillingInitialized := NOT Drilling.DeviceNotInitialized;
F_Drilling3 := Drilling.DeviceFault;

(* THINK DIAGNOSIS *)

FH_A_Drilling3 := Drilling.DeviceActuatorFaultHigh;
FL_A_Drilling3 := Drilling.DeviceActuatorFaultLow;


(*Block element Generic Device*)

Block(DeviceEnableRequest:=EnableBlock ,DeviceDisableRequest := DisableBlock);
A_BlockElement3 := Block.EnableDevice;
Block.DeviceType := DEVICE_WITH_SINGLE_ACTUATION OR DEVICE_WITHOUT_FEEDBACK;
Block.DeviceClock := ClocksGeneration.Clock2ms;
Block.DeviceDiagnosticsEnabled := TRUE;
Block.DeviceDisableTime := 20;
Block.DeviceEnablePreset := FALSE;
Block.DeviceEnableTime := 20;
Block.DeviceOperation := OperationType;
BlockInitialized := NOT Block.DeviceNotInitialized;
F_Block3 := Block.DeviceFault;

(* THINK DIAGNOSIS *)

FH_A_Block3 := Block.DeviceActuatorFaultHigh;
FL_A_Block3 := Block.DeviceActuatorFaultLow;


(*Expell Generic Device*)

Expell(DeviceEnableRequest:=EnableExpell ,DeviceDisableRequest := DisableExpell);
A_ExpellElement3 := Expell.EnableDevice;
Expell.DeviceType := DEVICE_WITH_SINGLE_ACTUATION OR DEVICE_WITHOUT_FEEDBACK;
Expell.DeviceClock := ClocksGeneration.Clock2ms;
Expell.DeviceDiagnosticsEnabled := TRUE;
Expell.DeviceDisableTime := 20;
Expell.DeviceEnablePreset := FALSE;
Expell.DeviceEnableTime := 20;
Expell.DeviceOperation := OperationType;
ExpellInitialized := NOT Expell.DeviceNotInitialized;
F_Expell3 := Expell.DeviceFault;

(* THINK DIAGNOSIS *)

FH_A_Expell3 := Expell.DeviceActuatorFaultHigh;
FL_A_Expell3 := Expell.DeviceActuatorFaultLow;
END_FUNCTION_BLOCK

(* POU Work_Station/S4, ST *)
FUNCTION_BLOCK S4

VAR_INPUT

	ElementColor: BOOL;
	ElementOver: BOOL;

END_VAR

VAR_OUTPUT

	InitializationDone4: BOOL := FALSE;
	GoS3:BOOL:=FALSE;
	RobotIsMoving:BOOL:=FALSE;
	RobotIsOn:BOOL:=FALSE;
	NotSafeToRestart: BOOL := FALSE;
	OnPhaseStopDone4: BOOL := FALSE;
	StopDone4: BOOL;
	Element: CharacterisazionElement;
	Idle:BOOL;
	Completed:INT:=0;
	Rejected:INT:=0;

END_VAR

VAR

	SpringExtractor:GenericDevice;
	PistonSelector: GenericDevice;
	ExtractCoverInAssemblyStation: GenericDevice;
	BlockingCylinder: GenericDevice;

	RobotInitPose: GenericDevice;
	RobotTakeBlack: GenericDevice;
	RobotTakeRed: GenericDevice;
	RobotDiscardBlack: GenericDevice;
	RobotDiscardRed: GenericDevice;
	RobotToAssembly: GenericDevice;
	RobotTakeSpring: GenericDevice;
	RobotTakePiston: GenericDevice;
	RobotTakeCover: GenericDevice;
	RobotReset: GenericDevice;

	EnableSpringExtractor: BOOL:=FALSE;
	EnablePistonSelector: BOOL:=FALSE;
	EnableExtractCoverInAssemblyStation: BOOL:=FALSE;
	EnableBlockingCylinder: BOOL:=FALSE;

	EnableRobotInitPose: BOOL:=FALSE;
	EnableRobotTakeBlack: BOOL:=FALSE;
	EnableRobotTakeRed: BOOL:=FALSE;
	EnableRobotDiscardBlack: BOOL:=FALSE;
	EnableRobotDiscardRed: BOOL:=FALSE;
	EnableRobotToAssembly: BOOL:=FALSE;
	EnableRobotTakeSpring: BOOL:=FALSE;
	EnableRobotTakePiston: BOOL:=FALSE;
	EnableRobotTakeCover: BOOL:=FALSE;
	EnableRobotReset: BOOL:=FALSE;


	DisableSpringExtractor: BOOL:=FALSE;
	DisablePistonSelector: BOOL:=FALSE;
	DisableExtractCoverInAssemblyStation: BOOL:=FALSE;
	DisableBlockingCylinder: BOOL:=FALSE;

	DisableRobotInitPose: BOOL := FALSE;
	DisableRobotTakeBlack: BOOL:=FALSE;
	DisableRobotTakeRed: BOOL:=FALSE;
	DisableRobotDiscardBlack: BOOL:=FALSE;
	DisableRobotDiscardRed: BOOL:=FALSE;
	DisableRobotToAssembly: BOOL:=FALSE;
	DisableRobotTakeSpring: BOOL:=FALSE;
	DisableRobotTakePiston: BOOL:=FALSE;
	DisableRobotTakeCover: BOOL:=FALSE;
	DisableRobotReset: BOOL:=FALSE;

	StateMachine: INT;
	State2Counter: INT := 2;
	SpringExtractorInitialized: BOOL := FALSE;
	PistonSelectorInitialized: BOOL := FALSE;
	ExtractCoverInAssemblyStationInitialized: BOOL := FALSE;
	BlockingCylinderInitialized: BOOL := FALSE;
	RobotInitialized: BOOL := FALSE;

END_VAR

VAR_IN_OUT

	OperationType: INT;

END_VAR
IF NOT S_ElementAvailable4 THEN

	GoS3 := TRUE;

ELSE

	GoS3:= FALSE;

END_IF

(*Number of spring*)

IF B_FillAll OR B_SpringLoader THEN

	NumSpring:=8;

END_IF

SpringHouseNotEmpty := NOT (NumSpring=0);

(*Number of piston*)

IF B_FillAll OR  B_PistonLoader THEN
	NumPistonBlack := 8;
	NumPistonGrey := 8;
END_IF
PistonHouseNotEmpty := NOT (NumPistonBlack=0 OR NumPistonGrey=0);

CASE OperationType OF

	INIT:

		IF SpringExtractorInitialized AND PistonSelectorInitialized AND ExtractCoverInAssemblyStationInitialized AND BlockingCylinderInitialized AND RobotInitialized AND NOT S_NoCover4 (*AND SpringHouseNotEmpty*) THEN
			InitializationDone4 := TRUE;
		END_IF

	READYTORUN:

		NotSafeToRestart := FALSE;
		StopOutput4 := FALSE;
		OnPhaseStopDone4 := FALSE;
		StopDone4 := FALSE;

	RUN:

		CASE StateMachine OF

			0: (*Reset the robot*)

				EnableRobotReset := TRUE;
				Idle:=TRUE;
				IF State2Counter > 0 THEN
					State2Counter := State2Counter -1;
				ELSE
					DisableRobotReset := TRUE;
					State2Counter := 2;
					StateMachine := 5;
				END_IF

			5: (*Depending on the element characterization choose the right command for the robot*)

				IF  S_ElementAvailable4 THEN
					Idle:=FALSE;
					Element.Color:=ElementColor;
					Element.Over:=ElementOver;
					RobotIsOn := TRUE;
					IF  Element.Over THEN (* PIece Overturned*)
						IF Element.Color THEN
							EnableRobotDiscardRed := TRUE;
							StateMachine := 75;
						ELSE
							EnableRobotDiscardBlack := TRUE;
							StateMachine := 80;
						END_IF
					ELSE (* If Fine *)
						IF Element.Color THEN
							EnableRobotTakeRed := TRUE;
							NumPistonBlack:=NumPistonBlack-1;
							StateMachine := 10;
						ELSE
							EnableRobotTakeBlack := TRUE;
							NumPistonGrey:=NumPistonGrey-1;
							StateMachine := 25;
						END_IF
					END_IF
				END_IF

			(*PROCEDURE FOR GOOD PIECES*)

			10: (*Pieces setup for assembly for Red/Silver elements up to state 20*)

				IF NOT EnableRobotTakeRed THEN
					DisableRobotTakeRed := TRUE;
					DisableBlockingCylinder:=TRUE;
					DisableSpringExtractor:=TRUE;
					EnableExtractCoverInAssemblyStation:=TRUE;
					EnablePistonSelector:=TRUE;
					StateMachine:=15;
				END_IF

			15:
				IF NOT DisableBlockingCylinder AND NOT DisableSpringExtractor  AND NOT EnableExtractCoverInAssemblyStation AND NOT EnablePistonSelector  THEN
					EnableSpringExtractor:=TRUE;
					DisablePistonSelector:=TRUE;
					DisableExtractCoverInAssemblyStation:=TRUE;
					StateMachine:=20;
				END_IF

			20:
				IF NOT EnableSpringExtractor AND NOT DisableExtractCoverInAssemblyStation AND NOT DisablePistonSelector THEN
					EnableRobotTakePiston := TRUE;
					StateMachine:=40;
				END_IF

			25: (*Pieces setup for assembly for Red/Silver elements up to state 35*)

				IF NOT EnableRobotTakeBlack THEN
					DisableRobotTakeBlack := TRUE;
					DisableBlockingCylinder:=TRUE;
					DisableSpringExtractor:=TRUE;
					EnableExtractCoverInAssemblyStation:=TRUE;
					DisablePistonSelector:=TRUE;
					StateMachine:=30;
				END_IF

			30:

				IF NOT DisableBlockingCylinder AND NOT DisableSpringExtractor  AND NOT EnableExtractCoverInAssemblyStation AND NOT DisablePistonSelector  THEN
					EnableSpringExtractor:=TRUE;
					EnablePistonSelector:=TRUE;
					DisableExtractCoverInAssemblyStation:=TRUE;
					StateMachine:=35;
				END_IF

			35:

				IF NOT EnableSpringExtractor AND NOT DisableExtractCoverInAssemblyStation AND NOT EnablePistonSelector THEN
					EnableRobotTakePiston := TRUE;
					StateMachine:=40;
				END_IF

			40: (*Take Piston*)

				IF NOT EnableRobotTakePiston THEN
					DisableRobotTakePiston := TRUE;
					EnableRobotToAssembly := TRUE;
					StateMachine:=45;
				END_IF

			45: (*Return to assembly*)

				IF NOT EnableRobotToAssembly THEN
					DisableRobotToAssembly := TRUE;
					EnableRobotTakeSpring := TRUE;
					NumSpring:=NumSpring-1;
					StateMachine:=50;
				END_IF

			50: (*Take Spring*)

				IF NOT EnableRobotTakeSpring THEN
					DisableRobotTakeSpring := TRUE;
					EnableRobotToAssembly := TRUE;
					StateMachine:=55;
				END_IF

			55: (*Return to assembly*)

				IF NOT EnableRobotToAssembly  THEN
					DisableRobotToAssembly := TRUE;
					IF NOT S_NoCover4 THEN
						EnableRobotTakeCover := TRUE;
						StateMachine:=60;
					END_IF
				END_IF

			60: (*Take Cover*)

				IF NOT EnableRobotTakeCover THEN
					DisableRobotTakeCover := TRUE;
					EnableRobotToAssembly := TRUE;
					StateMachine:=65;
				END_IF

			65: (*Return to assembly*)

				IF NOT EnableRobotToAssembly  THEN
					DisableRobotToAssembly := TRUE;
					EnableBlockingCylinder:=TRUE;
					StateMachine:=70;
				END_IF

			70: (*Piece completed*)

				IF NOT EnableBlockingCylinder THEN
					EnableRobotInitPose := TRUE;
					Completed:=Completed+1;
					StateMachine:=100;
				END_IF

			(*PROCEDURE FOR PIECES TO DISCARD*)

			75: (*Discard Red Piece*)

				IF NOT EnableRobotDiscardRed THEN
					Rejected:=Rejected+1;
					DisableRobotDiscardRed := TRUE;
					EnableRobotInitPose := TRUE;
					StateMachine := 100;
				END_IF

			80: (*Discard Black Piece*)

				IF NOT EnableRobotDiscardBlack THEN
					Rejected:=Rejected+1;
					DisableRobotDiscardBlack := TRUE;
					EnableRobotInitPose := TRUE;
					StateMachine := 100;
				END_IF

			100: (*Return to init position*)

				IF NOT EnableRobotInitPose THEN
					DisableRobotInitPose := TRUE;
					EnableRobotReset := TRUE;
					RobotIsOn := FALSE;
					StateMachine := 0;
				END_IF

		END_CASE

	IMMEDIATESTOPMACHINE:

		CASE StateMachine OF

			0:
				StopDone4 := TRUE;

			5:
				StopDone4 := TRUE;

			10:
				IF EnableRobotTakeRed THEN
					StopOutput4 := TRUE;
					NotSafeToRestart := TRUE;
				END_IF
				StopDone4 := TRUE;

			15:
				IF NOT DisableBlockingCylinder AND NOT DisableSpringExtractor  AND NOT EnableExtractCoverInAssemblyStation AND NOT EnablePistonSelector  THEN
					StopDone4 := TRUE;
				END_IF

			20:
				IF NOT EnableSpringExtractor AND NOT DisableExtractCoverInAssemblyStation AND NOT DisablePistonSelector THEN
					StopDone4 := TRUE;
				END_IF

			25:
				IF EnableRobotTakeBlack THEN
					StopOutput4 := TRUE;
					NotSafeToRestart := TRUE;
				END_IF
				StopDone4 := TRUE;

			30:
				IF NOT DisableBlockingCylinder AND NOT DisableSpringExtractor  AND NOT EnableExtractCoverInAssemblyStation AND NOT DisablePistonSelector  THEN
					StopDone4 := TRUE;
				END_IF

			35:
				IF NOT EnableSpringExtractor AND NOT DisableExtractCoverInAssemblyStation AND NOT EnablePistonSelector THEN
					StopDone4 := TRUE;
				END_IF

			40:
				IF EnableRobotTakePiston THEN
					StopOutput4 := TRUE;
					NotSafeToRestart := TRUE;
				END_IF
				StopDone4 := TRUE;

			45:
				IF EnableRobotToAssembly THEN
					StopOutput4 := TRUE;
					NotSafeToRestart := TRUE;
				END_IF
				StopDone4 := TRUE;

			50:
				IF EnableRobotTakeSpring THEN
					StopOutput4 := TRUE;
					NotSafeToRestart := TRUE;
				END_IF
				StopDone4 := TRUE;

			55:
				IF EnableRobotToAssembly  THEN
					StopOutput4 := TRUE;
					NotSafeToRestart := TRUE;
				END_IF
				StopDone4 := TRUE;

			60:
				IF EnableRobotTakeCover THEN
					StopOutput4 := TRUE;
					NotSafeToRestart := TRUE;
				END_IF
				StopDone4 := TRUE;

			65:
				IF EnableRobotToAssembly  THEN
					StopOutput4 := TRUE;
					NotSafeToRestart := TRUE;
				END_IF
				StopDone4 := TRUE;

			70:
				IF EnableBlockingCylinder THEN
					StopDone4 := TRUE;
				END_IF

			75:
				IF EnableRobotDiscardRed THEN
					StopOutput4 := TRUE;
					NotSafeToRestart := TRUE;
				END_IF
				StopDone4 := TRUE;

			80:
				IF EnableRobotDiscardBlack THEN
					StopOutput4 := TRUE;
					NotSafeToRestart := TRUE;
				END_IF
				StopDone4 := TRUE;

			100:
				IF EnableRobotInitPose THEN
					StopOutput4 := TRUE;
					NotSafeToRestart := TRUE;
				END_IF
				StopDone4 := TRUE;

		END_CASE

	ONPHASESTOPMACHINE:

		CASE StateMachine OF

			0:
				OnPhaseStopDone4 := TRUE;

			5:
				OnPhaseStopDone4 := TRUE;

			10:
				IF NOT EnableRobotTakeRed THEN
					OnPhaseStopDone4 := TRUE;
				END_IF

			15:
				IF NOT DisableBlockingCylinder AND NOT DisableSpringExtractor  AND NOT EnableExtractCoverInAssemblyStation AND NOT EnablePistonSelector  THEN
					OnPhaseStopDone4 := TRUE;
				END_IF

			20:
				IF NOT EnableSpringExtractor AND NOT DisableExtractCoverInAssemblyStation AND NOT DisablePistonSelector THEN
					OnPhaseStopDone4 := TRUE;
				END_IF

			25:
				IF NOT EnableRobotTakeBlack THEN
					OnPhaseStopDone4 := TRUE;
				END_IF

			30:
				IF NOT DisableBlockingCylinder AND NOT DisableSpringExtractor  AND NOT EnableExtractCoverInAssemblyStation AND NOT DisablePistonSelector  THEN
					OnPhaseStopDone4 := TRUE;
				END_IF

			35:
				IF NOT EnableSpringExtractor AND NOT DisableExtractCoverInAssemblyStation AND NOT EnablePistonSelector THEN
					OnPhaseStopDone4 := TRUE;
				END_IF

			40:
				IF NOT EnableRobotTakePiston THEN
					OnPhaseStopDone4 := TRUE;
				END_IF

			45:
				IF NOT EnableRobotToAssembly THEN
					OnPhaseStopDone4 := TRUE;
				END_IF

			50:
				IF NOT EnableRobotTakeSpring THEN
					OnPhaseStopDone4 := TRUE;
				END_IF

			55:
				IF NOT EnableRobotToAssembly  THEN
					OnPhaseStopDone4 := TRUE;
				END_IF

			60:
				IF NOT EnableRobotTakeCover THEN
					OnPhaseStopDone4 := TRUE;
				END_IF

			65:
				IF NOT EnableRobotToAssembly  THEN
					OnPhaseStopDone4 := TRUE;
				END_IF

			70:
				IF NOT EnableBlockingCylinder THEN
					OnPhaseStopDone4 := TRUE;
				END_IF

			75:
				IF NOT EnableRobotDiscardRed THEN
					OnPhaseStopDone4 := TRUE;
				END_IF

			80:
				IF NOT EnableRobotDiscardBlack THEN
					OnPhaseStopDone4 := TRUE;
				END_IF

			100:
				IF NOT EnableRobotInitPose THEN
					OnPhaseStopDone4 := TRUE;
				END_IF

			END_CASE

	READYTORESET:

		EnableRobotReset := TRUE;
		StopOutput4 := FALSE;
		StateMachine := 0;
		InitializationDone4 := FALSE;

END_CASE

(*SpringExtractor Generic Device*)

SpringExtractor(DeviceEnableRequest:=EnableSpringExtractor ,DeviceDisableRequest := DisableSpringExtractor);
A_SpringCylinder4 := SpringExtractor.EnableDevice;
SpringExtractor.DeviceEnabled := S_SpringCylinderRetracted4;
SpringExtractor.DeviceDisabled := S_SpringCylinderExtended4;
SpringExtractor.DeviceType := DEVICE_WITH_SINGLE_ACTUATION OR DEVICE_WITH_DOUBLE_FEEDBACK;
SpringExtractor.DeviceClock := ClocksGeneration.Clock2ms;
SpringExtractor.DeviceDiagnosticsEnabled := TRUE;
SpringExtractor.DeviceDisableTime := 30;
SpringExtractor.DeviceEnablePreset := TRUE;
SpringExtractor.DeviceEnableTime := 30;
SpringExtractorInitialized := NOT SpringExtractor.DeviceNotInitialized;
SpringExtractor.DeviceOperation := OperationType;
F_SpringExtractor4 := SpringExtractor.DeviceFault;
F_S_SpringExtractor4 := SpringExtractor.DeviceSensorFault;
F_A_SpringExtractor4 := SpringExtractor.DeviceActuatorFault;
FH_A_SpringExtractor4 := SpringExtractor.DeviceActuatorFaultHigh;
FL_A_SpringExtractor4 := SpringExtractor.DeviceActuatorFaultLow;
FH_DS_SpringExtractor4 := SpringExtractor.DeviceEnabledSensorFaultHigh;
FL_DS_SpringExtractor4 := SpringExtractor.DeviceEnabledSensorFaultLow;
FH_ES_SpringExtractor4 := SpringExtractor.DeviceDisabledSensorFaultHigh;
FL_ES_SpringExtractor4 := SpringExtractor.DeviceDisabledSensorFaultLow;

(*Piston Selector Generic Device*)

PistonSelector(DeviceEnableRequest:=EnablePistonSelector ,DeviceDisableRequest := DisablePistonSelector);
A_GiveBlackPiston4 := PistonSelector.EnableDevice;
A_GiveSilverPiston4 := PistonSelector.DisableDevice;
PistonSelector.DeviceEnabled := S_BlackPistonGiven4;
PistonSelector.DeviceDisabled := S_SilverPistonGiven4;
PistonSelector.DeviceType := DEVICE_WITH_DOUBLE_ACTUATION OR DEVICE_WITH_DOUBLE_FEEDBACK;
PistonSelector.DeviceClock := ClocksGeneration.Clock2ms;
PistonSelector.DeviceDiagnosticsEnabled := TRUE;
PistonSelector.DeviceDisableTime := 30;
PistonSelector.DeviceEnablePreset := FALSE;
PistonSelector.DeviceEnableTime := 30;
PistonSelectorInitialized := NOT PistonSelector.DeviceNotInitialized;
PistonSelector.DeviceOperation := OperationType;
F_PistonSelector4 := PistonSelector.DeviceFault;
F_S_PistonSelector4 := PistonSelector.DeviceSensorFault;
F_A_PistonSelector4 := PistonSelector.DeviceActuatorFault;
FH_EA_PistonSelector4 := PistonSelector.DeviceEnableActuatorFaultHigh;
FL_EA_PistonSelector4 := PistonSelector.DeviceEnableActuatorFaultLow;
FH_DA_PistonSelector4 := PistonSelector.DeviceDisableActuatorFaultHigh;
FL_DA_PistonSelector4 := PistonSelector.DeviceDisableActuatorFaultLow;
FH_ES_PistonSelector4 := PistonSelector.DeviceEnabledSensorFaultHigh;
FL_ES_PistonSelector4 := PistonSelector.DeviceEnabledSensorFaultLow;
FH_DS_PistonSelector4 := PistonSelector.DeviceDisabledSensorFaultHigh;
FH_DS_PistonSelector4 := PistonSelector.DeviceDisabledSensorFaultLow;

(*Cover extractor Generic Device*)

ExtractCoverInAssemblyStation(DeviceEnableRequest:=EnableExtractCoverInAssemblyStation ,DeviceDisableRequest := DisableExtractCoverInAssemblyStation);
A_CoverCylinder4 := ExtractCoverInAssemblyStation.EnableDevice;
ExtractCoverInAssemblyStation.DeviceEnabled := S_CoverCylinderExtracted4;
ExtractCoverInAssemblyStation.DeviceDisabled := S_CoverCylinderRetracted4;
ExtractCoverInAssemblyStation.DeviceType := DEVICE_WITH_SINGLE_ACTUATION OR DEVICE_WITH_DOUBLE_FEEDBACK;
ExtractCoverInAssemblyStation.DeviceClock := ClocksGeneration.Clock2ms;
ExtractCoverInAssemblyStation.DeviceDiagnosticsEnabled := TRUE;
ExtractCoverInAssemblyStation.DeviceDisableTime := 30;
ExtractCoverInAssemblyStation.DeviceEnablePreset := TRUE;
ExtractCoverInAssemblyStation.DeviceEnableTime := 30;
ExtractCoverInAssemblyStationInitialized := NOT ExtractCoverInAssemblyStation.DeviceNotInitialized;
ExtractCoverInAssemblyStation.DeviceOperation := OperationType;
F_ExtractCover4 := ExtractCoverInAssemblyStation.DeviceFault;
F_S_ExtractCover4 := ExtractCoverInAssemblyStation.DeviceSensorFault;
F_A_ExtractCover4 := ExtractCoverInAssemblyStation.DeviceActuatorFault;
FH_A_ExtractCover4 := ExtractCoverInAssemblyStation.DeviceActuatorFaultHigh;
FL_A_ExtractCover4 := ExtractCoverInAssemblyStation.DeviceActuatorFaultLow;
FH_ES_ExtractCover4 := ExtractCoverInAssemblyStation.DeviceEnabledSensorFaultHigh;
FL_ES_ExtractCover4 := ExtractCoverInAssemblyStation.DeviceEnabledSensorFaultLow;
FH_DS_ExtractCover4 := ExtractCoverInAssemblyStation.DeviceDisabledSensorFaultHigh;
FL_DS_ExtractCover4 := ExtractCoverInAssemblyStation.DeviceDisabledSensorFaultLow;

(*Blocking cylinder Generic Device*)

BlockingCylinder(DeviceEnableRequest:=EnableBlockingCylinder ,DeviceDisableRequest := DisableBlockingCylinder);
A_BlockElement4 := BlockingCylinder.EnableDevice;
BlockingCylinder.DeviceType := DEVICE_WITH_SINGLE_ACTUATION OR DEVICE_WITHOUT_FEEDBACK;
BlockingCylinder.DeviceClock := ClocksGeneration.Clock2ms;
BlockingCylinder.DeviceDiagnosticsEnabled := TRUE;
BlockingCylinder.DeviceDisableTime := 30;
BlockingCylinder.DeviceEnablePreset := TRUE;
BlockingCylinder.DeviceEnableTime := 30;
BlockingCylinderInitialized := NOT BlockingCylinder.DeviceNotInitialized;
BlockingCylinder.DeviceOperation := OperationType;
F_BlockingCylinder4 := BlockingCylinder.DeviceFault;

(* THINK DIAGNOSIS *)

FH_A_BlockingCylinder4 := BlockingCylinder.DeviceActuatorFaultHigh;
FL_A_BlockingCylinder4 := BlockingCylinder.DeviceActuatorFaultLow;

(*Robot to Initial Position Generic Device*)

RobotInitPose(DeviceEnableRequest:=EnableRobotInitPose ,DeviceDisableRequest := DisableRobotInitPose);
A_RobotToInitial4 := RobotInitPose.EnableDevice;
RobotInitPose.DeviceEnabled := S_RobotInInitial4;
RobotInitPose.DeviceType := DEVICE_WITH_SINGLE_ACTUATION OR DEVICE_WITH_ENABLE_FEEDBACK;
RobotInitPose.DeviceClock := ClocksGeneration.Clock2ms;
RobotInitPose.DeviceDiagnosticsEnabled := TRUE;
RobotInitPose.DeviceDisableTime := 2;
RobotInitPose.DeviceEnablePreset := TRUE;
RobotInitPose.DeviceEnableTime := 200;
RobotInitPose.DeviceOperation := OperationType;
RobotInitialized := NOT RobotInitPose.DeviceNotInitialized;
F_A_RobotToInitial4 := RobotInitPose.DeviceActuatorFault;
F_S_RobotInInitial4 := RobotInitPose.DeviceEnabledSensorFault;

(*Robot take a black piece Generic Device*)

RobotTakeBlack(DeviceEnableRequest:=EnableRobotTakeBlack ,DeviceDisableRequest := DisableRobotTakeBlack);
A_RobotTakeBlack4 := RobotTakeBlack.EnableDevice;
RobotTakeBlack.DeviceEnabled := S_RobotAssembly4;
RobotTakeBlack.DeviceType := DEVICE_WITH_SINGLE_ACTUATION OR DEVICE_WITH_ENABLE_FEEDBACK;
RobotTakeBlack.DeviceClock := ClocksGeneration.Clock2ms;
RobotTakeBlack.DeviceDiagnosticsEnabled := TRUE;
RobotTakeBlack.DeviceDisableTime := 2;
RobotTakeBlack.DeviceEnablePreset := FALSE;
RobotTakeBlack.DeviceEnableTime := 200;
RobotTakeBlack.DeviceOperation := OperationType;

(*Robot take a red/silver piece Generic Device*)

RobotTakeRed(DeviceEnableRequest:=EnableRobotTakeRed ,DeviceDisableRequest := DisableRobotTakeRed);
A_RobotTakeRedSilver4 := RobotTakeRed.EnableDevice;
RobotTakeRed.DeviceEnabled := S_RobotAssembly4;
RobotTakeRed.DeviceType := DEVICE_WITH_SINGLE_ACTUATION OR DEVICE_WITH_ENABLE_FEEDBACK;
RobotTakeRed.DeviceClock := ClocksGeneration.Clock2ms;
RobotTakeRed.DeviceDiagnosticsEnabled := TRUE;
RobotTakeRed.DeviceDisableTime := 2;
RobotTakeRed.DeviceEnablePreset := FALSE;
RobotTakeRed.DeviceEnableTime := 200;
RobotTakeRed.DeviceOperation := OperationType;

(*Robot discard a black piece Generic Device*)

RobotDiscardBlack(DeviceEnableRequest:=EnableRobotDiscardBlack ,DeviceDisableRequest := DisableRobotDiscardBlack);
A_RobotDiscardBlack4 := RobotDiscardBlack.EnableDevice;
RobotDiscardBlack.DeviceEnabled := S_RobotInInitial4;
RobotDiscardBlack.DeviceType := DEVICE_WITH_SINGLE_ACTUATION OR DEVICE_WITH_ENABLE_FEEDBACK;
RobotDiscardBlack.DeviceClock := ClocksGeneration.Clock2ms;
RobotDiscardBlack.DeviceDiagnosticsEnabled := TRUE;
RobotDiscardBlack.DeviceDisableTime := 2;
RobotDiscardBlack.DeviceEnablePreset := FALSE;
RobotDiscardBlack.DeviceEnableTime := 200;
RobotDiscardBlack.DeviceOperation := OperationType;

(*Robot discard a red/silver piece Generic Device*)

RobotDiscardRed(DeviceEnableRequest:=EnableRobotDiscardRed ,DeviceDisableRequest := DisableRobotDiscardRed);
A_RobotDiscardRedSilver4 := RobotDiscardRed.EnableDevice;
RobotDiscardRed.DeviceEnabled := S_RobotInInitial4;
RobotDiscardRed.DeviceType := DEVICE_WITH_SINGLE_ACTUATION OR DEVICE_WITH_ENABLE_FEEDBACK;
RobotDiscardRed.DeviceClock := ClocksGeneration.Clock2ms;
RobotDiscardRed.DeviceDiagnosticsEnabled := TRUE;
RobotDiscardRed.DeviceDisableTime := 2;
RobotDiscardRed.DeviceEnablePreset := FALSE;
RobotDiscardRed.DeviceEnableTime := 200;
RobotDiscardRed.DeviceOperation := OperationType;

(*Robot go to Assembly*)

RobotToAssembly(DeviceEnableRequest:=EnableRobotToAssembly ,DeviceDisableRequest := DisableRobotToAssembly);
A_RobotAssembly4 := RobotToAssembly.EnableDevice;
RobotToAssembly.DeviceEnabled := S_RobotAssembly4;
RobotToAssembly.DeviceType := DEVICE_WITH_SINGLE_ACTUATION OR DEVICE_WITH_ENABLE_FEEDBACK;
RobotToAssembly.DeviceClock := ClocksGeneration.Clock2ms;
RobotToAssembly.DeviceDiagnosticsEnabled := TRUE;
RobotToAssembly.DeviceDisableTime := 2;
RobotToAssembly.DeviceEnablePreset := FALSE;
RobotToAssembly.DeviceEnableTime := 250;
RobotToAssembly.DeviceOperation := OperationType;
F_A_RobotAssembly4 := RobotToAssembly.DeviceActuatorFault;
F_S_RobotAssembly4 := RobotToAssembly.DeviceEnabledSensorFault;

(*Robot take a spring Generic Device*)

RobotTakeSpring(DeviceEnableRequest:=EnableRobotTakeSpring ,DeviceDisableRequest := DisableRobotTakeSpring);
A_RobotSpring4 := RobotTakeSpring.EnableDevice;
RobotTakeSpring.DeviceEnabled := S_RobotSpring4;
RobotTakeSpring.DeviceType := DEVICE_WITH_SINGLE_ACTUATION OR DEVICE_WITH_ENABLE_FEEDBACK;
RobotTakeSpring.DeviceClock := ClocksGeneration.Clock2ms;
RobotTakeSpring.DeviceDiagnosticsEnabled := TRUE;
RobotTakeSpring.DeviceDisableTime := 2;
RobotTakeSpring.DeviceEnablePreset := FALSE;
RobotTakeSpring.DeviceEnableTime := 200;
RobotTakeSpring.DeviceOperation := OperationType;
F_A_RobotSpring4 := RobotTakeSpring.DeviceActuatorFault;
F_S_RobotSpring4 := RobotTakeSpring.DeviceEnabledSensorFault;

(*Robot take a piston Generic Device*)

RobotTakePiston(DeviceEnableRequest:=EnableRobotTakePiston ,DeviceDisableRequest := DisableRobotTakePiston);
A_RobotPiston4 := RobotTakePiston.EnableDevice;
RobotTakePiston.DeviceEnabled := S_RobotPiston4;
RobotTakePiston.DeviceType := DEVICE_WITH_SINGLE_ACTUATION OR DEVICE_WITH_ENABLE_FEEDBACK;
RobotTakePiston.DeviceClock := ClocksGeneration.Clock2ms;
RobotTakePiston.DeviceDiagnosticsEnabled := TRUE;
RobotTakePiston.DeviceDisableTime := 2;
RobotTakePiston.DeviceEnablePreset := FALSE;
RobotTakePiston.DeviceEnableTime := 200;
RobotTakePiston.DeviceOperation := OperationType;
F_A_RobotPiston4 := RobotTakePiston.DeviceActuatorFault;
F_S_RobotPiston4 := RobotTakePiston.DeviceEnabledSensorFault;

(*Robot take a cover Generic Device*)

RobotTakeCover(DeviceEnableRequest:=EnableRobotTakeCover ,DeviceDisableRequest := DisableRobotTakeCover);
A_RobotCover4 := RobotTakeCover.EnableDevice;
RobotTakeCover.DeviceEnabled := S_RobotCover4;
RobotTakeCover.DeviceType := DEVICE_WITH_SINGLE_ACTUATION OR DEVICE_WITH_ENABLE_FEEDBACK;
RobotTakeCover.DeviceClock := ClocksGeneration.Clock2ms;
RobotTakeCover.DeviceDiagnosticsEnabled := TRUE;
RobotTakeCover.DeviceDisableTime := 2;
RobotTakeCover.DeviceEnablePreset := FALSE;
RobotTakeCover.DeviceEnableTime := 200;
RobotTakeCover.DeviceOperation := OperationType;
F_A_RobotCover4 := RobotTakeCover.DeviceActuatorFault;
F_S_RobotCover4 := RobotTakeCover.DeviceEnabledSensorFault;

(*Robot Reset Generic Device*)

RobotReset(DeviceEnableRequest:=EnableRobotReset ,DeviceDisableRequest := DisableRobotReset);
A_RobotReset4 := RobotReset.EnableDevice;
RobotReset.DeviceEnabled := S_RobotInInitial4;
RobotReset.DeviceType := DEVICE_WITH_SINGLE_ACTUATION OR DEVICE_WITH_ENABLE_FEEDBACK;
RobotReset.DeviceClock := ClocksGeneration.Clock2ms;
RobotReset.DeviceDiagnosticsEnabled := TRUE;
RobotReset.DeviceDisableTime := 2;
RobotReset.DeviceEnablePreset := FALSE;
RobotReset.DeviceEnableTime := 200;
RobotReset.DeviceOperation := OperationType;

(*Robot control part*)

IF NOT S_RobotInInitial4 AND NOT S_RobotCover4 AND NOT S_RobotPiston4 AND NOT S_RobotSpring4 AND NOT S_RobotAssembly4 THEN
	RobotIsMoving := TRUE;
ELSE
	RobotIsMoving := FALSE;
END_IF
END_FUNCTION_BLOCK

(* POU Lights, ST *)
FUNCTION_BLOCK Lights

VAR_INPUT

	InitializationDone:BOOL;
	OperationType:INT;
	RobotMoving: BOOL;
	RobotOn: BOOL;
	Element2: CharacterisazionElement;
	Element3: CharacterisazionElement;
	Element4: CharacterisazionElement;
	PieceToDiscard2 : BOOL;
	WriteLight2:BOOL;
	WriteLight3: BOOL;
	WriteLight4: BOOL;
	Completed:INT;
	Rejected:INT;

END_VAR

VAR_OUTPUT

END_VAR

VAR

END_VAR
CASE OperationType OF

	INIT:

		L_Reset := FALSE;
		VL_StateReset:=FALSE;

		VL_StateInit := TRUE;

	READYTORUN:

		VL_StateInit := FALSE;
		VL_StateImmediateStop := FALSE;
		VL_StateStop := FALSE;

		VL_StateReady := TRUE;
		L_Start := NOT L_Start;

	RUN:

		VL_StateReady := FALSE;

		L_Start := TRUE;
		VL_StateRun := TRUE;

		IF WriteLight2 THEN
			IF Element2.Color  THEN
				VL_ColorVis2 :=16#0000FF;  (*Red/Silver Piece*)
			ELSE
				VL_ColorVis2 := 16#000000; (*Black Piece*)
			END_IF
		ELSE
				VL_ColorVis2 := 16#FFFFFF; (*White if no pieces are present *)
		END_IF

		IF WriteLight3 THEN
			IF Element3.Color  THEN
				VL_ColorVis :=16#0000FF; (*Red/Silver Piece*)
			ELSE
				VL_ColorVis := 16#000000; (*Black Piece*)
			END_IF
			IF Element3.Over THEN
				VL_PositionVis := 16#FF0000; (*Blue if it is overturned *)
			ELSE
				VL_PositionVis :=16#00FF00; (*Green if it is on the right side*)
			END_IF
		ELSE
				VL_ColorVis := 16#FFFFFF; (*White if no pieces are present *)
				VL_PositionVis := 16#FFFFFF; (*White if no pieces are present *)
		END_IF

		IF WriteLight4 THEN
			IF Element4.Color  THEN
				VL_ColorVis4 :=16#0000FF; (*Red/Silver Piece*)
			ELSE
				VL_ColorVis4 := 16#000000; (*Black Piece*)
			END_IF
		ELSE
				VL_ColorVis4 := 16#FFFFFF; (*White if no pieces are present *)
		END_IF

		VL_Completed:=Completed;
		VL_Rejected:=Rejected;

		(*Red/Silver element loaded*)
		IF RobotOn AND  Element4.Color THEN
			L_RedSilverElement := TRUE;
		ELSE
			L_RedSilverElement := FALSE;
		END_IF

		(*Black element loaded*)
		IF RobotOn AND NOT  Element4.Color THEN
			L_BlackElement := TRUE;
		ELSE
			L_BlackElement := FALSE;
		END_IF

		(*Overturned element light in station 4*)
		IF  RobotOn AND Element4.Over THEN
			L_UpsideDownElement := TRUE;
		ELSE
			L_UpsideDownElement := FALSE;
		END_IF

		(* Piece with uncorrect height*)
		IF PieceToDiscard2 THEN
			L_PieceToDiscard2 := TRUE;
		ELSE
			L_PieceToDiscard2 := FALSE;
		END_IF

	IMMEDIATESTOPMACHINE:

		L_Start := FALSE;
		VL_StateRun := FALSE;
		L_RedSilverElement := FALSE;
		L_BlackElement := FALSE;
		L_UpsideDownElement := FALSE;
		VL_StateReady := FALSE;

		VL_StateImmediateStop := TRUE;

	ONPHASESTOPMACHINE:

		L_Start := FALSE;
		VL_StateRun := FALSE;
		L_RedSilverElement := FALSE;
		L_BlackElement := FALSE;
		L_UpsideDownElement := FALSE;
		VL_StateReady := FALSE;

		VL_StateStop := TRUE;

	EMERGENCYSTOPMACHINE:

		L_Start := FALSE;
		VL_StateRun := FALSE;
		L_RedSilverElement := FALSE;
		L_BlackElement := FALSE;
		L_UpsideDownElement := FALSE;
		VL_StateReady := FALSE;

		VL_StateAlarm := TRUE;

	READYTORESET:

		VL_StateImmediateStop := FALSE;
		VL_StateAlarm:=FALSE;

		VL_StateReset:=TRUE;
		L_Reset := NOT L_Reset;

END_CASE

(*Emptywarehouse light*)
IF S_EmptyWarehouse1 THEN
	L_EmptyWarehouse := TRUE;
ELSE
	L_EmptyWarehouse := FALSE;
END_IF

(*Deposit with no cover*)
IF S_NoCover4 THEN
	L_NoCover := TRUE;
ELSE
	L_NoCover := FALSE;
END_IF

(*Robot moving*)
IF RobotMoving AND RobotOn THEN
	L_RobotMoving := TRUE;
ELSE
	L_RobotMoving := FALSE;
END_IF

(*Robot ON*)
IF RobotOn THEN
	L_RobotOn := TRUE;
ELSE
	L_RobotOn := FALSE;
END_IF
END_FUNCTION_BLOCK

(* POU SignalHandler, ST *)
PROGRAM SignalHandler

VAR

	SignalManagement : SignalManagement;
	BaseAlarm : INT;
	BaseAnomaly : INT;

END_VAR
(* Update reset Inputs not dependant from signal *)

SignalManagement.ResetSignal := (FaultRemoved OR FaultDetected);
SignalManagement.KeyReset := KeyReset;
SignalManagement.CumulativeReset := CumulativeReset;

(* OUTPUT EXECUTION *)

TypeOfFault := PrioritySignalToString(SignalManagement.SignalPriorityCode);

(* Update Fault History, only if signal has generated an output *)

IF NOT (SignalManagement.SignalPriorityCode = SignalPriorityCode1) AND NOT (SignalManagement.SignalOutputs = NONE) THEN
	SignalPriorityCode3 := SignalPriorityCode2;
	SignalPriorityCode2 := SignalPriorityCode1;
	SignalPriorityCode1 := SignalManagement.SignalPriorityCode;
END_IF

TypeOfFault1 := PrioritySignalToString(SignalPriorityCode1); TypeOfFault2 := PrioritySignalToString(SignalPriorityCode2); TypeOfFault3 := PrioritySignalToString(SignalPriorityCode3);

(* Update Reset Condition and Fault flags *)

IF (SignalManagement.SignalOutputs = NONE) THEN
	NoSignalsToReset := TRUE;		(* Machine Reset Enabled only if no active outputs *)
	PossibleFault := FALSE;			(* Used for HMI *)
	Fault := FALSE;					(* Used for HMI *)
ELSE
	NoSignalsToReset := FALSE;
	PossibleFault := TRUE;
	Fault:= TRUE;
END_IF

(* Update Output Commands for Controller *)

EmergencyInStop := ((SignalManagement.SignalOutputs AND EMERGENCY_STOP) = EMERGENCY_STOP) OR B_Emergency;
ImmediateInStop := ((SignalManagement.SignalOutputs AND IMMEDIATE_STOP) = IMMEDIATE_STOP);
OnPhaseInStop := ((SignalManagement.SignalOutputs AND ON_PHASE_STOP) = ON_PHASE_STOP);

(* PERFORM INIT or RUN Operations *)

IF (SignHandlerOperationType = INIT) THEN
	SignalManagement.OperationType := INIT;
	SignalManagement();
	SignalManagement.OperationType := START_CONFIGURATION;
	SignalManagement();
	SignalManagement.OperationType := CONFIGURATION;
ELSE
	SignalManagement.OperationType := START_GENERATION;
	SignalManagement();
	SignalManagement.OperationType := GENERATION;
END_IF;

(* Big List of SIGNAL CALLS SimulationPlant Dependant *)

SignalManagement.SignalType := ALARM + AUX_RESET;
SignalManagement.SignalCode := mEmergencyButtonPressed;
SignalManagement.SignalOutput := EMERGENCY_STOP;
SignalManagement.ActivationSignal := B_Emergency;
SignalManagement.AutoResetSignal := NOT B_Emergency;
SignalManagement();

SignalManagement.SignalType := ALARM + AUTO_CONDITIONED_RESET;
SignalManagement.SignalCode := mFreezeButtonPressed;
SignalManagement.SignalOutput := IMMEDIATE_STOP;
SignalManagement.ActivationSignal := B_Freeze;
SignalManagement.AutoResetSignal := NOT B_Freeze;
SignalManagement();

SignalManagement.SignalType := ALARM + AUTO_CONDITIONED_RESET;
SignalManagement.SignalCode := mOnPhaseStopButtonPressed;
SignalManagement.SignalOutput := ON_PHASE_STOP;
SignalManagement.ActivationSignal := B_Stop;
SignalManagement.AutoResetSignal := NOT B_Stop;
SignalManagement();

SignalManagement.SignalType := WARNING + AUTO_CONDITIONED_RESET + AUTO_PROVISIONAL_RESET;
SignalManagement.ProvisionalDelay := WaitingTime * 10;
SignalManagement.SignalCode := mIdleStopAutoRequest ;
SignalManagement.SignalOutput :=ON_PHASE_STOP;
SignalManagement.ActivationSignal := AllStationsIdle;
SignalManagement.AutoResetSignal := NOT AllStationsIdle ;
SignalManagement();

SignalManagement.SignalType := INFORMATION + AUTO_CONDITIONED_RESET ;
SignalManagement.SignalCode := mEmptyWarehouse ;
SignalManagement.SignalOutput :=NONE;
SignalManagement.ActivationSignal := S_EmptyWarehouse1;
SignalManagement.AutoResetSignal := NOT S_EmptyWarehouse1;
SignalManagement();

SignalManagement.SignalType := INFORMATION + AUTO_CONDITIONED_RESET ;
SignalManagement.SignalCode := mEmpyCoverInAssembly;
SignalManagement.SignalOutput :=NONE;
SignalManagement.ActivationSignal := S_NoCover4;
SignalManagement.AutoResetSignal := NOT S_NoCover4 ;
SignalManagement();

(**********************************************************************************************)

IF SensorActuationDiagnosticEnabled THEN

SignalManagement.SignalType := ALARM + AUTO_CONDITIONED_RESET + AUTO_PROVISIONAL_RESET;
SignalManagement.ProvisionalDelay := OUTPUT_COUNTER_DELAY;
SignalManagement.SignalCode := mS1CylinderActuationFault;
SignalManagement.SignalOutput := IMMEDIATE_STOP;
SignalManagement.ActivationSignal := F_A_Cylinder1;
SignalManagement.AutoResetSignal := NOT F_A_Cylinder1 ;
SignalManagement();

SignalManagement.SignalType := ALARM + AUTO_CONDITIONED_RESET + AUTO_PROVISIONAL_RESET;
SignalManagement.ProvisionalDelay := OUTPUT_COUNTER_DELAY;
SignalManagement.SignalCode := mS1ArmActuationFault;
SignalManagement.SignalOutput := IMMEDIATE_STOP;
SignalManagement.ActivationSignal := F_A_Rotary1;
SignalManagement.AutoResetSignal := NOT F_A_Rotary1;
SignalManagement();

SignalManagement.SignalType := ALARM + AUTO_CONDITIONED_RESET + AUTO_PROVISIONAL_RESET;
SignalManagement.ProvisionalDelay := OUTPUT_COUNTER_DELAY;
SignalManagement.SignalCode := mS1VacuumActuationFault;
SignalManagement.SignalOutput := IMMEDIATE_STOP;
SignalManagement.ActivationSignal := F_A_Vacuum1;
SignalManagement.AutoResetSignal := NOT F_A_Vacuum1;
SignalManagement();
(*
SignalManagement.SignalType := ALARM + AUTO_CONDITIONED_RESET + AUTO_PROVISIONAL_RESET;
SignalManagement.ProvisionalDelay := OUTPUT_COUNTER_DELAY;
SignalManagement.SignalCode := mS2ElevatorActuationFault;
SignalManagement.SignalOutput := IMMEDIATE_STOP;
SignalManagement.ActivationSignal := F_A_Elevator2;
SignalManagement.AutoResetSignal := NOT F_A_Elevator2;
SignalManagement();
*)
SignalManagement.SignalType := ALARM + AUTO_CONDITIONED_RESET + AUTO_PROVISIONAL_RESET;
SignalManagement.ProvisionalDelay := OUTPUT_COUNTER_DELAY;
SignalManagement.SignalCode := mS2CylinderActuationFault;
SignalManagement.SignalOutput := IMMEDIATE_STOP;
SignalManagement.ActivationSignal := F_A_Cylinder2;
SignalManagement.AutoResetSignal := NOT F_A_Cylinder2;
SignalManagement();

SignalManagement.SignalType := ALARM + AUTO_CONDITIONED_RESET + AUTO_PROVISIONAL_RESET;
SignalManagement.ProvisionalDelay := OUTPUT_COUNTER_DELAY;
SignalManagement.SignalCode := mS3RotaryActuationFault;
SignalManagement.SignalOutput := IMMEDIATE_STOP;
SignalManagement.ActivationSignal := F_A_RotaryTable3;
SignalManagement.AutoResetSignal := NOT F_A_RotaryTable3;
SignalManagement();

SignalManagement.SignalType := ALARM + AUTO_CONDITIONED_RESET + AUTO_PROVISIONAL_RESET;
SignalManagement.ProvisionalDelay := OUTPUT_COUNTER_DELAY;
SignalManagement.SignalCode := mS3DrillCylinderActuationFault;
SignalManagement.SignalOutput := IMMEDIATE_STOP;
SignalManagement.ActivationSignal := F_A_DrillCylinder3;
SignalManagement.AutoResetSignal := NOT F_A_DrillCylinder3;
SignalManagement();

SignalManagement.SignalType := ALARM + AUTO_CONDITIONED_RESET + AUTO_PROVISIONAL_RESET;
SignalManagement.ProvisionalDelay := OUTPUT_COUNTER_DELAY;
SignalManagement.SignalCode := mS4SpringExtractorActuationFault;
SignalManagement.SignalOutput := IMMEDIATE_STOP;
SignalManagement.ActivationSignal := F_A_SpringExtractor4;
SignalManagement.AutoResetSignal := NOT F_A_SpringExtractor4;
SignalManagement();

SignalManagement.SignalType := ALARM + AUTO_CONDITIONED_RESET + AUTO_PROVISIONAL_RESET;
SignalManagement.ProvisionalDelay := OUTPUT_COUNTER_DELAY;
SignalManagement.SignalCode := mS4PistonSelectorActuationFault;
SignalManagement.SignalOutput := IMMEDIATE_STOP;
SignalManagement.ActivationSignal := F_A_PistonSelector4;
SignalManagement.AutoResetSignal := NOT F_A_PistonSelector4;
SignalManagement();

SignalManagement.SignalType := ALARM + AUTO_CONDITIONED_RESET + AUTO_PROVISIONAL_RESET;
SignalManagement.ProvisionalDelay := OUTPUT_COUNTER_DELAY;
SignalManagement.SignalCode := mS4CoverExtractorActuationFault;
SignalManagement.SignalOutput := IMMEDIATE_STOP;
SignalManagement.ActivationSignal := F_A_ExtractCover4;
SignalManagement.AutoResetSignal := NOT F_A_ExtractCover4;
SignalManagement();
(*
SignalManagement.SignalType := ALARM + AUTO_CONDITIONED_RESET + AUTO_PROVISIONAL_RESET;
SignalManagement.ProvisionalDelay := OUTPUT_COUNTER_DELAY;;
SignalManagement.SignalCode := mS4RobotInitActuationFault;
SignalManagement.SignalOutput := IMMEDIATE_STOP;
SignalManagement.ActivationSignal := F_A_RobotToInitial4;
SignalManagement.AutoResetSignal := NOT F_A_RobotToInitial4;
SignalManagement();
*)
SignalManagement.SignalType := ALARM + AUTO_CONDITIONED_RESET + AUTO_PROVISIONAL_RESET;
SignalManagement.ProvisionalDelay := OUTPUT_COUNTER_DELAY;
SignalManagement.SignalCode := mS4RobotPistonActuationFault;
SignalManagement.SignalOutput := IMMEDIATE_STOP;
SignalManagement.ActivationSignal := F_A_RobotPiston4;
SignalManagement.AutoResetSignal := NOT F_A_RobotPiston4;
SignalManagement();

SignalManagement.SignalType := ALARM + AUTO_CONDITIONED_RESET + AUTO_PROVISIONAL_RESET;
SignalManagement.ProvisionalDelay := OUTPUT_COUNTER_DELAY;
SignalManagement.SignalCode := mS4RobotSpringActuationFault;
SignalManagement.SignalOutput := IMMEDIATE_STOP;
SignalManagement.ActivationSignal := F_A_RobotSpring4;
SignalManagement.AutoResetSignal := NOT F_A_RobotSpring4;
SignalManagement();

SignalManagement.SignalType := ALARM + AUTO_CONDITIONED_RESET + AUTO_PROVISIONAL_RESET;
SignalManagement.ProvisionalDelay := OUTPUT_COUNTER_DELAY;
SignalManagement.SignalCode := mS4RobotCoverActuationFault;
SignalManagement.SignalOutput := IMMEDIATE_STOP;
SignalManagement.ActivationSignal := F_A_RobotCover4;
SignalManagement.AutoResetSignal := NOT F_A_RobotCover4;
SignalManagement();
(*
SignalManagement.SignalType := ALARM + AUTO_CONDITIONED_RESET + AUTO_PROVISIONAL_RESET;
SignalManagement.ProvisionalDelay := OUTPUT_COUNTER_DELAY;
SignalManagement.SignalCode := mS4RobotAssemblyActuationFault;
SignalManagement.SignalOutput := IMMEDIATE_STOP;
SignalManagement.ActivationSignal := F_A_RobotAssembly4;
SignalManagement.AutoResetSignal := NOT F_A_RobotAssembly4;
SignalManagement();
*)
SignalManagement.SignalType := ANOMALY + AUTO_CONDITIONED_RESET + AUTO_PROVISIONAL_RESET;
SignalManagement.ProvisionalDelay := OUTPUT_COUNTER_DELAY;
SignalManagement.SignalCode := mS1CylinderSensorFault;
SignalManagement.SignalOutput := ON_PHASE_STOP;
SignalManagement.ActivationSignal := F_S_Cylinder1;
SignalManagement.AutoResetSignal := NOT F_S_Cylinder1;
SignalManagement();

SignalManagement.SignalType := ANOMALY + AUTO_CONDITIONED_RESET + AUTO_PROVISIONAL_RESET;
SignalManagement.ProvisionalDelay := OUTPUT_COUNTER_DELAY;
SignalManagement.SignalCode := mS1ArmSensorFault;
SignalManagement.SignalOutput := ON_PHASE_STOP;
SignalManagement.ActivationSignal := F_S_Rotary1;
SignalManagement.AutoResetSignal := NOT F_S_Rotary1;
SignalManagement();

SignalManagement.SignalType := ANOMALY + AUTO_CONDITIONED_RESET + AUTO_PROVISIONAL_RESET;
SignalManagement.ProvisionalDelay := OUTPUT_COUNTER_DELAY;
SignalManagement.SignalCode := mS1VacuumSensorFault;
SignalManagement.SignalOutput := ON_PHASE_STOP;
SignalManagement.ActivationSignal := F_S_Vacuum1;
SignalManagement.AutoResetSignal := NOT F_S_Vacuum1;
SignalManagement();
(*
SignalManagement.SignalType := ANOMALY + AUTO_CONDITIONED_RESET + AUTO_PROVISIONAL_RESET;
SignalManagement.ProvisionalDelay := OUTPUT_COUNTER_DELAY;
SignalManagement.SignalCode := mS2ElevatorSensorFault;
SignalManagement.SignalOutput := ON_PHASE_STOP;
SignalManagement.ActivationSignal := F_S_Elevator2;
SignalManagement.AutoResetSignal := NOT F_S_Elevator2;
SignalManagement();
*)
SignalManagement.SignalType := ANOMALY + AUTO_CONDITIONED_RESET + AUTO_PROVISIONAL_RESET;
SignalManagement.ProvisionalDelay := OUTPUT_COUNTER_DELAY;
SignalManagement.SignalCode := mS2CylinderSensorFault;
SignalManagement.SignalOutput := ON_PHASE_STOP;
SignalManagement.ActivationSignal := F_S_Cylinder2;
SignalManagement.AutoResetSignal := NOT F_S_Cylinder2;
SignalManagement();

SignalManagement.SignalType := ANOMALY + AUTO_CONDITIONED_RESET + AUTO_PROVISIONAL_RESET;
SignalManagement.ProvisionalDelay := OUTPUT_COUNTER_DELAY;
SignalManagement.SignalCode := mS3RotarySensorFault;
SignalManagement.SignalOutput := NONE;
SignalManagement.ActivationSignal := F_S_RotaryTable3;
SignalManagement.AutoResetSignal := NOT F_S_RotaryTable3;
SignalManagement();

SignalManagement.SignalType := ANOMALY + AUTO_CONDITIONED_RESET + AUTO_PROVISIONAL_RESET;
SignalManagement.ProvisionalDelay := OUTPUT_COUNTER_DELAY;
SignalManagement.SignalCode := mS3DrillCylinderSensorFault;
SignalManagement.SignalOutput := ON_PHASE_STOP;
SignalManagement.ActivationSignal := F_S_DrillCylinder3;
SignalManagement.AutoResetSignal := NOT F_S_DrillCylinder3;
SignalManagement();

SignalManagement.SignalType := ANOMALY + AUTO_CONDITIONED_RESET + AUTO_PROVISIONAL_RESET;
SignalManagement.ProvisionalDelay := OUTPUT_COUNTER_DELAY;
SignalManagement.SignalCode := mS4SpringExtractorSensorFault;
SignalManagement.SignalOutput := ON_PHASE_STOP;
SignalManagement.ActivationSignal := F_S_SpringExtractor4;
SignalManagement.AutoResetSignal := NOT F_S_SpringExtractor4;
SignalManagement();

SignalManagement.SignalType := ANOMALY + AUTO_CONDITIONED_RESET + AUTO_PROVISIONAL_RESET;
SignalManagement.ProvisionalDelay := OUTPUT_COUNTER_DELAY;
SignalManagement.SignalCode := mS4PistonSelectorSensorFault;
SignalManagement.SignalOutput := ON_PHASE_STOP;
SignalManagement.ActivationSignal := F_S_PistonSelector4;
SignalManagement.AutoResetSignal := NOT F_S_PistonSelector4;
SignalManagement();

SignalManagement.SignalType := ANOMALY + AUTO_CONDITIONED_RESET + AUTO_PROVISIONAL_RESET;
SignalManagement.ProvisionalDelay := OUTPUT_COUNTER_DELAY;
SignalManagement.SignalCode := mS4CoverExtractorSensorFault;
SignalManagement.SignalOutput := ON_PHASE_STOP;
SignalManagement.ActivationSignal := F_S_ExtractCover4;
SignalManagement.AutoResetSignal := NOT F_S_ExtractCover4;
SignalManagement();
(*
SignalManagement.SignalType := ANOMALY + AUTO_CONDITIONED_RESET + AUTO_PROVISIONAL_RESET;
SignalManagement.ProvisionalDelay := OUTPUT_COUNTER_DELAY;
SignalManagement.SignalCode := mS4RobotInitSensorFault;
SignalManagement.SignalOutput := ON_PHASE_STOP;
SignalManagement.ActivationSignal := F_S_RobotInInitial4;
SignalManagement.AutoResetSignal := NOT F_S_RobotInInitial4;
SignalManagement();
*)
SignalManagement.SignalType := ANOMALY + AUTO_CONDITIONED_RESET + AUTO_PROVISIONAL_RESET;
SignalManagement.ProvisionalDelay := OUTPUT_COUNTER_DELAY;
SignalManagement.SignalCode := mS4RobotPistonSensorFault;
SignalManagement.SignalOutput := ON_PHASE_STOP;
SignalManagement.ActivationSignal := F_S_RobotPiston4;
SignalManagement.AutoResetSignal := NOT F_S_RobotPiston4;
SignalManagement();

SignalManagement.SignalType := ANOMALY + AUTO_CONDITIONED_RESET + AUTO_PROVISIONAL_RESET;
SignalManagement.ProvisionalDelay := OUTPUT_COUNTER_DELAY;
SignalManagement.SignalCode := mS4RobotSpringSensorFault;
SignalManagement.SignalOutput := ON_PHASE_STOP;
SignalManagement.ActivationSignal := F_S_RobotSpring4;
SignalManagement.AutoResetSignal := NOT F_S_RobotSpring4;
SignalManagement();

SignalManagement.SignalType := ANOMALY + AUTO_CONDITIONED_RESET + AUTO_PROVISIONAL_RESET;
SignalManagement.ProvisionalDelay := OUTPUT_COUNTER_DELAY;
SignalManagement.SignalCode := mS4RobotCoverSensorFault;
SignalManagement.SignalOutput := ON_PHASE_STOP;
SignalManagement.ActivationSignal := F_S_RobotCover4;
SignalManagement.AutoResetSignal := NOT F_S_RobotCover4;
SignalManagement();

SignalManagement.SignalType := ANOMALY + AUTO_CONDITIONED_RESET + AUTO_PROVISIONAL_RESET;
SignalManagement.ProvisionalDelay := OUTPUT_COUNTER_DELAY;
SignalManagement.SignalCode := mS4RobotAssemblySensorFault;
SignalManagement.SignalOutput := ON_PHASE_STOP;
SignalManagement.ActivationSignal := F_S_RobotAssembly4;
SignalManagement.AutoResetSignal := NOT F_S_RobotAssembly4;
SignalManagement();

END_IF
END_PROGRAM

(* POU MyLibraries/SignalManagement, ST *)
FUNCTION_BLOCK SignalManagement

VAR_INPUT

	OperationType : INT;			(* Configurazione della libreria *)
	SignalType : WORD;			(* Tipo di segnale e tipo di Reset *)
	SignalCode : WORD;			(* Codice segnale *)
	SignalOutput : DWORD;		(* Output desiderato se segnale attivo *)
	ActivationSignal : BOOL;		(* Segnale di attivazione *)
	AutoResetSignal : BOOL := FALSE;		(* Segnale per attivare condizione autoreset *)
	KeyReset : BOOL := FALSE;		(* To link KEY-VAR for AuxReset *)
	ResetSignal : BOOL := FALSE;	(* Signal To do Reset *)
	CumulativeReset: BOOL := FALSE; (* IF TRUE cumulative reset is performed *)
	ProvisionalDelay: INT ;

END_VAR

VAR_OUTPUT

	SignalOutputs : DWORD;		(* Output Attivi, Immediate or OnPhase or Emergency *)
	SignalPriorityCode : WORD;	(* Segnale attivo con più alta priorità, se 0 è nullo *)
	ResetEnable : BOOL;			(* Segnale abilitato al reset *)
	AuxResetEnable : BOOL;

END_VAR

VAR_EXTERNAL

	INIT : INT :=1;
	START_CONFIGURATION : INT := 12;
	CONFIGURATION : INT := 13;
	START_GENERATION : INT := 14;
	GENERATION : INT := 15;

 (* BitMask for Signal Type *)

	ALARM : WORD := 00001;
	ANOMALY : WORD := 00002;
	WARNING : WORD := 00003;
	INFORMATION : WORD := 00004;
	SIGNAL_TYPE_MASK : WORD := 00007;

(* BitMasks for Reset types *)

	AUX_RESET : WORD := 512;			 (* Reset enabled only if aux reset input active *)
	AUTO_RESET : WORD := 1024;		(*Reset  IF ActivationSignal is not present anymore *)
	AUTO_CONDITIONED_RESET : WORD := 2048;	(* Reset IF ActivatSignal not pres anymore AND IF AutoResetSignal TRUE *)
	UNCONDITIONED_RESET : WORD := 4096;		(* Reset in any case if most important *)
	AUTO_PROVISIONAL_RESET : WORD := 8192;		(* Dont Activate If ProvisionalDelay not Expired *)

	AUTO_PRIORITY_RESET : WORD := 16384;

	(* SignalOutputs *)

	NONE : DWORD := 16#000;
	EMERGENCY_STOP : DWORD := 16#0001;
	IMMEDIATE_STOP : DWORD := 16#0002;
	ON_PHASE_STOP : DWORD := 16#0004;

END_VAR

